C05474=1196.791,200.391,-58.412,-177.682,6.514,148.507
C05475=1196.796,200.142,-58.389,-177.685,6.512,148.508
C05476=1196.800,199.893,-58.365,-177.688,6.510,148.508
C05477=1196.805,199.644,-58.342,-177.690,6.508,148.508
C05478=1196.809,199.396,-58.317,-177.692,6.506,148.509
C05479=1196.813,199.146,-58.294,-177.695,6.505,148.509
C05480=1196.818,198.898,-58.270,-177.698,6.502,148.509
C05481=1196.823,198.649,-58.246,-177.701,6.500,148.510
C05482=1196.827,198.400,-58.222,-177.704,6.498,148.510
C05483=1196.832,198.151,-58.199,-177.706,6.497,148.510
C05484=1196.836,197.902,-58.175,-177.709,6.495,148.511
C05485=1196.841,197.653,-58.151,-177.712,6.493,148.511
C05486=1196.846,197.404,-58.127,-177.714,6.491,148.511
C05487=1196.851,197.155,-58.104,-177.716,6.489,148.511
C05488=1196.855,196.907,-58.080,-177.719,6.487,148.512
C05489=1196.860,196.658,-58.057,-177.722,6.485,148.512
C05490=1196.864,196.409,-58.033,-177.724,6.484,148.512
C05491=1196.869,196.160,-58.009,-177.727,6.482,148.513
C05492=1196.874,195.911,-57.986,-177.730,6.480,148.513
C05493=1196.878,195.662,-57.963,-177.732,6.478,148.514
C05494=1196.883,195.414,-57.938,-177.735,6.476,148.514
C05495=1196.888,195.165,-57.915,-177.738,6.475,148.514
C05496=1196.892,194.916,-57.892,-177.740,6.473,148.515
C05497=1196.896,194.668,-57.868,-177.743,6.471,148.515
C05498=1196.901,194.419,-57.845,-177.745,6.469,148.515
C05499=1196.905,194.170,-57.822,-177.748,6.467,148.515
C05500=1196.910,193.921,-57.798,-177.751,6.465,148.516
C05501=1196.914,193.672,-57.774,-177.753,6.463,148.516
C05502=1196.919,193.423,-57.751,-177.756,6.462,148.516
C05503=1196.924,193.174,-57.727,-177.759,6.460,148.517
C05504=1196.929,192.925,-57.704,-177.761,6.458,148.517
C05505=1196.933,192.676,-57.681,-177.764,6.456,148.517
C05506=1196.938,192.427,-57.657,-177.766,6.454,148.518
C05507=1196.942,192.179,-57.633,-177.769,6.452,148.518
C05508=1196.947,191.930,-57.610,-177.772,6.451,148.519
C05509=1196.951,191.681,-57.587,-177.774,6.449,148.519
C05510=1196.956,191.433,-57.564,-177.777,6.447,148.519
C05511=1196.961,191.184,-57.541,-177.780,6.445,148.520
C05512=1196.966,190.935,-57.517,-177.782,6.443,148.520
C05513=1196.970,190.685,-57.494,-177.785,6.441,148.520
C05514=1196.975,190.436,-57.471,-177.787,6.439,148.520
C05515=1196.979,190.188,-57.448,-177.790,6.438,148.521
C05516=1196.984,189.939,-57.425,-177.793,6.436,148.521
C05517=1196.988,189.690,-57.401,-177.795,6.434,148.521
C05518=1196.993,189.441,-57.378,-177.798,6.432,148.522
C05519=1196.998,189.192,-57.354,-177.801,6.430,148.522
C05520=1197.003,188.943,-57.331,-177.803,6.429,148.523
C05521=1197.007,188.695,-57.309,-177.806,6.427,148.523
C05522=1197.012,188.446,-57.285,-177.809,6.425,148.523
C05523=1197.016,188.196,-57.262,-177.811,6.423,148.524
C05524=1197.021,187.947,-57.239,-177.814,6.421,148.524
C05525=1197.025,187.699,-57.216,-177.817,6.420,148.524
C05526=1197.030,187.450,-57.193,-177.819,6.418,148.525
C05527=1197.035,187.201,-57.169,-177.822,6.416,148.525
C05528=1197.040,186.952,-57.146,-177.825,6.414,148.525
C05529=1197.044,186.704,-57.123,-177.827,6.412,148.526
C05530=1197.049,186.455,-57.100,-177.830,6.411,148.526
C05531=1197.053,186.206,-57.077,-177.833,6.409,148.526
C05532=1197.057,185.957,-57.054,-177.835,6.407,148.527
C05533=1197.062,185.708,-57.031,-177.838,6.405,148.527
C05534=1197.067,185.459,-57.008,-177.841,6.403,148.527
C05535=1197.072,185.189,-56.984,-177.843,6.402,148.528
C05536=1197.077,184.920,-56.958,-177.846,6.400,148.528
C05537=1197.082,184.650,-56.933,-177.849,6.397,148.528
C05538=1197.087,184.381,-56.909,-177.852,6.395,148.529
C05539=1197.092,184.132,-56.885,-177.854,6.394,148.529
C05540=1197.096,183.883,-56.863,-177.857,6.392,148.530
C05541=1197.101,183.634,-56.840,-177.860,6.390,148.530
C05542=1197.105,183.385,-56.817,-177.862,6.388,148.530
C05543=1197.110,183.137,-56.794,-177.864,6.387,148.531
C05544=1197.115,182.887,-56.771,-177.867,6.385,148.531
C05545=1197.120,182.638,-56.748,-177.870,6.384,148.531
C05546=1197.124,182.389,-56.725,-177.872,6.382,148.532
C05547=1197.129,182.140,-56.703,-177.875,6.380,148.532
C05548=1197.133,181.892,-56.680,-177.878,6.378,148.532
C05549=1197.138,181.642,-56.657,-177.880,6.376,148.533
C05550=1197.142,181.394,-56.634,-177.883,6.375,148.533
C05551=1197.147,181.145,-56.612,-177.886,6.373,148.534
C05552=1197.151,180.896,-56.589,-177.888,6.371,148.534
C05553=1197.156,180.647,-56.566,-177.891,6.369,148.534
C05554=1197.161,180.397,-56.543,-177.894,6.367,148.535
C05555=1197.166,180.149,-56.521,-177.896,6.366,148.535
C05556=1197.171,179.900,-56.498,-177.899,6.364,148.535
C05557=1197.175,179.651,-56.475,-177.902,6.362,148.536
C05558=1197.180,179.403,-56.452,-177.904,6.361,148.536
C05559=1197.184,179.153,-56.430,-177.907,6.359,148.537
C05560=1197.189,178.904,-56.407,-177.910,6.358,148.537
C05561=1197.193,178.655,-56.385,-177.912,6.356,148.537
C05562=1197.198,178.407,-56.362,-177.915,6.354,148.538
C05563=1197.203,178.157,-56.340,-177.918,6.352,148.538
C05564=1197.207,177.909,-56.317,-177.920,6.350,148.538
C05565=1197.212,177.660,-56.295,-177.923,6.349,148.539
C05566=1197.216,177.411,-56.272,-177.926,6.347,148.539
C05567=1197.221,177.161,-56.249,-177.928,6.345,148.539
C05568=1197.226,176.913,-56.227,-177.931,6.343,148.540
C05569=1197.231,176.664,-56.204,-177.933,6.342,148.540
C05570=1197.235,176.415,-56.182,-177.936,6.341,148.541
C05571=1197.240,176.166,-56.160,-177.938,6.339,148.541
C05572=1197.244,175.917,-56.137,-177.941,6.337,148.541
C05573=1197.249,175.669,-56.115,-177.944,6.335,148.542
C05574=1197.254,175.419,-56.092,-177.946,6.333,148.542
C05575=1197.258,175.170,-56.069,-177.949,6.332,148.542
C05576=1197.263,174.922,-56.048,-177.952,6.330,148.543
C05577=1197.268,174.672,-56.024,-177.954,6.328,148.543
C05578=1197.272,174.423,-56.002,-177.957,6.326,148.543
C05579=1197.277,174.175,-55.981,-177.959,6.325,148.544
C05580=1197.282,173.925,-55.957,-177.962,6.324,148.544
C05581=1197.286,173.677,-55.936,-177.965,6.322,148.545
C05582=1197.291,173.427,-55.914,-177.968,6.320,148.545
C05583=1197.295,173.178,-55.890,-177.970,6.318,148.546
C05584=1197.300,172.930,-55.869,-177.973,6.317,148.546
C05585=1197.305,172.680,-55.847,-177.976,6.315,148.546
C05586=1197.310,172.432,-55.824,-177.978,6.313,148.547
C05587=1197.314,172.183,-55.801,-177.980,6.312,148.547
C05588=1197.319,171.934,-55.780,-177.983,6.310,148.547
C05589=1197.324,171.685,-55.757,-177.986,6.308,148.548
C05590=1197.328,171.436,-55.734,-177.989,6.307,148.548
C05591=1197.333,171.187,-55.713,-177.991,6.305,148.548
C05592=1197.337,170.938,-55.691,-177.994,6.303,148.549
C05593=1197.343,170.689,-55.668,-177.997,6.301,148.549
C05594=1197.347,170.440,-55.646,-177.999,6.301,148.550
C05595=1197.352,170.192,-55.624,-178.002,6.299,148.550
C05596=1197.356,169.942,-55.602,-178.004,6.297,148.551
C05597=1197.361,169.693,-55.580,-178.007,6.295,148.551
C05598=1197.366,169.444,-55.558,-178.010,6.293,148.551
C05599=1197.371,169.195,-55.536,-178.012,6.292,148.552
C05600=1197.375,168.946,-55.514,-178.015,6.290,148.552
C05601=1197.379,168.698,-55.491,-178.017,6.289,148.552
C05602=1197.384,168.448,-55.469,-178.020,6.287,148.553
C05603=1197.389,168.200,-55.447,-178.023,6.285,148.553
C05604=1197.394,167.950,-55.425,-178.025,6.283,148.553
C05605=1197.398,167.702,-55.403,-178.028,6.282,148.554
C05606=1197.403,167.452,-55.381,-178.031,6.280,148.554
C05607=1197.408,167.204,-55.360,-178.034,6.278,148.555
C05608=1197.413,166.954,-55.337,-178.036,6.277,148.555
C05609=1197.417,166.705,-55.315,-178.039,6.276,148.556
C05610=1197.422,166.456,-55.293,-178.041,6.274,148.556
C05611=1197.427,166.207,-55.272,-178.044,6.272,148.556
C05612=1197.431,165.958,-55.250,-178.047,6.270,148.557
C05613=1197.436,165.709,-55.228,-178.049,6.268,148.557
C05614=1197.440,165.460,-55.206,-178.052,6.268,148.558
C05615=1197.445,165.211,-55.184,-178.054,6.266,148.558
C05616=1197.449,164.962,-55.162,-178.057,6.264,148.558
C05617=1197.455,164.713,-55.140,-178.060,6.262,148.559
C05618=1197.460,164.464,-55.118,-178.062,6.261,148.559
C05619=1197.464,164.215,-55.096,-178.065,6.260,148.559
C05620=1197.469,163.966,-55.074,-178.067,6.258,148.560
C05621=1197.473,163.717,-55.052,-178.070,6.256,148.560
C05622=1197.478,163.468,-55.031,-178.073,6.255,148.561
C05623=1197.482,163.219,-55.009,-178.076,6.253,148.561
C05624=1197.487,162.970,-54.988,-178.078,6.251,148.562
C05625=1197.492,162.721,-54.966,-178.081,6.250,148.562
C05626=1197.496,162.472,-54.944,-178.083,6.248,148.562
C05627=1197.501,162.223,-54.922,-178.086,6.247,148.563
C05628=1197.506,161.974,-54.900,-178.089,6.245,148.563
C05629=1197.510,161.725,-54.878,-178.092,6.243,148.564
C05630=1197.515,161.477,-54.857,-178.094,6.242,148.564
C05631=1197.520,161.227,-54.835,-178.096,6.241,148.564
C05632=1197.525,160.978,-54.814,-178.099,6.239,148.565
C05633=1197.530,160.729,-54.792,-178.102,6.237,148.565
C05634=1197.534,160.480,-54.770,-178.105,6.235,148.566
C05635=1197.539,160.231,-54.749,-178.107,6.234,148.566
C05636=1197.544,159.982,-54.727,-178.110,6.233,148.567
C05637=1197.548,159.733,-54.705,-178.112,6.231,148.567
C05638=1197.552,159.484,-54.684,-178.115,6.229,148.567
C05639=1197.558,159.215,-54.661,-178.118,6.227,148.568
C05640=1197.563,158.946,-54.638,-178.121,6.226,148.568
C05641=1197.568,158.677,-54.614,-178.124,6.224,148.569
C05642=1197.573,158.408,-54.591,-178.126,6.222,148.569
C05643=1197.577,158.160,-54.570,-178.129,6.221,148.569
C05644=1197.582,157.910,-54.548,-178.132,6.220,148.570
C05645=1197.587,157.661,-54.527,-178.134,6.218,148.570
C05646=1197.592,157.412,-54.506,-178.137,6.216,148.571
C05647=1197.596,157.162,-54.484,-178.140,6.215,148.571
C05648=1197.601,156.914,-54.462,-178.142,6.214,148.571
C05649=1197.606,156.665,-54.441,-178.144,6.212,148.572
C05650=1197.610,156.416,-54.420,-178.148,6.210,148.572
C05651=1197.615,156.167,-54.398,-178.150,6.209,148.573
C05652=1197.620,155.918,-54.377,-178.152,6.208,148.573
C05653=1197.625,155.669,-54.355,-178.155,6.206,148.574
C05654=1197.629,155.419,-54.334,-178.158,6.204,148.574
C05655=1197.634,155.170,-54.312,-178.160,6.202,148.574
C05656=1197.639,154.921,-54.292,-178.163,6.202,148.575
C05657=1197.643,154.673,-54.270,-178.166,6.200,148.575
C05658=1197.648,154.423,-54.249,-178.168,6.198,148.576
C05659=1197.653,154.174,-54.227,-178.171,6.196,148.576
C05660=1197.657,153.925,-54.207,-178.173,6.195,148.576
C05661=1197.662,153.677,-54.185,-178.176,6.194,148.577
C05662=1197.667,153.427,-54.164,-178.179,6.192,148.577
C05663=1197.672,153.178,-54.142,-178.182,6.190,148.578
C05664=1197.677,152.929,-54.121,-178.184,6.189,148.578
C05665=1197.681,152.680,-54.100,-178.186,6.188,148.579
C05666=1197.686,152.431,-54.079,-178.190,6.186,148.579
C05667=1197.690,152.182,-54.057,-178.192,6.184,148.580
C05668=1197.695,151.933,-54.037,-178.194,6.184,148.580
C05669=1197.700,151.684,-54.016,-178.197,6.182,148.580
C05670=1197.705,151.435,-53.994,-178.200,6.180,148.581
C05671=1197.710,151.186,-53.973,-178.203,6.178,148.581
C05672=1197.714,150.937,-53.951,-178.205,6.178,148.582
C05673=1197.719,150.687,-53.931,-178.208,6.176,148.582
C05674=1197.724,150.438,-53.910,-178.210,6.174,148.582
C05675=1197.728,150.190,-53.888,-178.213,6.172,148.583
C05676=1197.733,149.941,-53.868,-178.216,6.172,148.583
C05677=1197.738,149.691,-53.847,-178.218,6.170,148.584
C05678=1197.742,149.442,-53.825,-178.221,6.168,148.584
C05679=1197.747,149.193,-53.804,-178.223,6.167,148.585
C05680=1197.752,148.944,-53.784,-178.226,6.166,148.585
C05681=1197.757,148.695,-53.763,-178.229,6.164,148.586
C05682=1197.762,148.446,-53.741,-178.232,6.162,148.586
C05683=1197.766,148.197,-53.721,-178.234,6.161,148.586
C05684=1197.771,147.948,-53.700,-178.237,6.160,148.587
C05685=1197.775,147.698,-53.679,-178.240,6.158,148.587
C05686=1197.780,147.450,-53.657,-178.242,6.157,148.588
C05687=1197.785,147.200,-53.636,-178.244,6.155,148.588
C05688=1197.790,146.951,-53.616,-178.247,6.153,148.588
C05689=1197.795,146.702,-53.595,-178.250,6.152,148.589
C05690=1197.799,146.454,-53.574,-178.252,6.151,148.589
C05691=1197.804,146.205,-53.553,-178.255,6.149,148.590
C05692=1197.808,145.956,-53.533,-178.258,6.147,148.590
C05693=1197.814,145.706,-53.512,-178.260,6.147,148.591
C05694=1197.818,145.456,-53.490,-178.263,6.145,148.591
C05695=1197.823,145.207,-53.470,-178.266,6.143,148.592
C05696=1197.828,144.958,-53.449,-178.268,6.142,148.592
C05697=1197.832,144.710,-53.428,-178.271,6.141,148.593
C05698=1197.837,144.461,-53.407,-178.274,6.139,148.593
C05699=1197.842,144.212,-53.387,-178.276,6.138,148.593
C05700=1197.847,143.962,-53.366,-178.278,6.136,148.594
C05701=1197.851,143.713,-53.345,-178.282,6.135,148.594
C05702=1197.856,143.465,-53.325,-178.284,6.133,148.595
C05703=1197.861,143.215,-53.304,-178.286,6.132,148.595
C05704=1197.865,142.966,-53.283,-178.289,6.130,148.596
C05705=1197.870,142.717,-53.263,-178.292,6.129,148.596
C05706=1197.875,142.468,-53.242,-178.294,6.128,148.597
C05707=1197.880,142.219,-53.221,-178.297,6.126,148.597
C05708=1197.884,141.970,-53.201,-178.300,6.124,148.597
C05709=1197.890,141.721,-53.180,-178.302,6.124,148.598
C05710=1197.894,141.472,-53.159,-178.305,6.122,148.598
C05711=1197.898,141.222,-53.139,-178.308,6.120,148.599
C05712=1197.903,140.973,-53.118,-178.310,6.120,148.599
C05713=1197.908,140.724,-53.097,-178.313,6.118,148.600
C05714=1197.913,140.475,-53.076,-178.316,6.116,148.600
C05715=1197.917,140.226,-53.056,-178.318,6.115,148.601
C05716=1197.922,139.977,-53.036,-178.321,6.114,148.601
C05717=1197.927,139.727,-53.015,-178.324,6.112,148.602
C05718=1197.931,139.478,-52.994,-178.326,6.111,148.602
C05719=1197.936,139.230,-52.974,-178.329,6.110,148.603
C05720=1197.942,138.980,-52.954,-178.332,6.108,148.603
C05721=1197.946,138.731,-52.934,-178.334,6.107,148.603
C05722=1197.951,138.482,-52.913,-178.336,6.105,148.604
C05723=1197.956,138.233,-52.892,-178.339,6.105,148.604
C05724=1197.960,137.984,-52.872,-178.342,6.103,148.605
C05725=1197.965,137.735,-52.852,-178.344,6.101,148.605
C05726=1197.970,137.486,-52.831,-178.347,6.100,148.606
C05727=1197.975,137.236,-52.811,-178.350,6.099,148.606
C05728=1197.979,136.988,-52.791,-178.352,6.097,148.606
C05729=1197.984,136.738,-52.770,-178.354,6.096,148.607
C05730=1197.989,136.489,-52.749,-178.358,6.094,148.608
C05731=1197.993,136.240,-52.730,-178.360,6.093,148.608
C05732=1197.998,135.991,-52.709,-178.362,6.092,148.608
C05733=1198.003,135.742,-52.688,-178.366,6.090,148.609
C05734=1198.007,135.493,-52.668,-178.368,6.089,148.609
C05735=1198.012,135.243,-52.648,-178.370,6.088,148.610
C05736=1198.017,134.994,-52.628,-178.374,6.086,148.610
C05737=1198.022,134.745,-52.607,-178.376,6.085,148.611
C05738=1198.027,134.497,-52.587,-178.378,6.083,148.611
C05739=1198.032,134.247,-52.567,-178.382,6.082,148.612
C05740=1198.036,133.998,-52.547,-178.384,6.081,148.612
C05741=1198.040,133.749,-52.527,-178.386,6.079,148.613
C05742=1198.046,133.499,-52.506,-178.388,6.078,148.613
C05743=1198.050,133.231,-52.484,-178.392,6.077,148.614
C05744=1198.056,132.962,-52.463,-178.394,6.075,148.614
C05745=1198.061,132.694,-52.441,-178.398,6.074,148.615
C05746=1198.066,132.425,-52.419,-178.400,6.072,148.615
C05747=1198.071,132.176,-52.399,-178.403,6.071,148.616
C05748=1198.076,131.927,-52.379,-178.406,6.070,148.616
C05749=1198.080,131.678,-52.359,-178.408,6.068,148.616
C05750=1198.085,131.428,-52.339,-178.411,6.067,148.617
C05751=1198.091,131.180,-52.319,-178.413,6.065,148.617
C05752=1198.095,130.930,-52.299,-178.416,6.064,148.618
C05753=1198.100,130.681,-52.279,-178.419,6.063,148.618
C05754=1198.104,130.432,-52.259,-178.421,6.061,148.619
C05755=1198.109,130.183,-52.239,-178.424,6.060,148.619
C05756=1198.113,129.934,-52.218,-178.427,6.059,148.620
C05757=1198.119,129.685,-52.199,-178.429,6.058,148.620
C05758=1198.123,129.436,-52.179,-178.432,6.056,148.621
C05759=1198.128,129.186,-52.159,-178.435,6.055,148.621
C05760=1198.133,128.936,-52.139,-178.437,6.054,148.622
C05761=1198.138,128.687,-52.118,-178.440,6.052,148.622
C05762=1198.143,128.439,-52.099,-178.442,6.051,148.623
C05763=1198.148,128.190,-52.079,-178.445,6.050,148.623
C05764=1198.152,127.940,-52.059,-178.447,6.049,148.624
C05765=1198.157,127.691,-52.039,-178.450,6.047,148.624
C05766=1198.162,127.442,-52.019,-178.453,6.046,148.624
C05767=1198.167,127.193,-51.999,-178.455,6.045,148.625
C05768=1198.171,126.944,-51.979,-178.458,6.043,148.625
C05769=1198.176,126.694,-51.960,-178.460,6.042,148.626
C05770=1198.180,126.445,-51.939,-178.463,6.041,148.626
C05771=1198.186,126.196,-51.920,-178.466,6.040,148.627
C05772=1198.191,125.947,-51.900,-178.468,6.038,148.627
C05773=1198.195,125.698,-51.880,-178.471,6.037,148.628
C05774=1198.200,125.448,-51.860,-178.474,6.036,148.628
C05775=1198.205,125.199,-51.841,-178.477,6.034,148.629
C05776=1198.209,124.950,-51.821,-178.479,6.033,148.629
C05777=1198.214,124.701,-51.801,-178.482,6.032,148.630
C05778=1198.220,124.452,-51.782,-178.484,6.031,148.630
C05779=1198.224,124.203,-51.761,-178.487,6.029,148.631
C05780=1198.228,123.954,-51.742,-178.490,6.028,148.631
C05781=1198.233,123.704,-51.723,-178.492,6.027,148.632
C05782=1198.238,123.455,-51.703,-178.495,6.025,148.632
C05783=1198.243,123.206,-51.683,-178.497,6.024,148.633
C05784=1198.247,122.957,-51.663,-178.500,6.023,148.633
C05785=1198.253,122.708,-51.644,-178.502,6.022,148.634
C05786=1198.257,122.458,-51.624,-178.505,6.020,148.634
C05787=1198.262,122.209,-51.604,-178.508,6.020,148.635
C05788=1198.267,121.961,-51.585,-178.510,6.018,148.635
C05789=1198.272,121.711,-51.565,-178.513,6.017,148.636
C05790=1198.276,121.462,-51.546,-178.516,6.015,148.636
C05791=1198.281,121.213,-51.527,-178.519,6.014,148.637
C05792=1198.286,120.963,-51.507,-178.521,6.013,148.637
C05793=1198.290,120.714,-51.487,-178.524,6.011,148.637
C05794=1198.296,120.466,-51.467,-178.526,6.011,148.638
C05795=1198.300,120.216,-51.448,-178.529,6.009,148.639
C05796=1198.305,119.967,-51.429,-178.531,6.008,148.639
C05797=1198.310,119.718,-51.409,-178.534,6.007,148.640
C05798=1198.315,119.468,-51.390,-178.536,6.006,148.640
C05799=1198.319,119.219,-51.370,-178.539,6.004,148.641
C05800=1198.325,118.970,-51.351,-178.542,6.003,148.641
C05801=1198.329,118.720,-51.331,-178.545,6.002,148.642
C05802=1198.334,118.472,-51.312,-178.547,6.001,148.642
C05803=1198.338,118.223,-51.292,-178.550,5.999,148.642
C05804=1198.343,117.973,-51.272,-178.552,5.999,148.643
C05805=1198.349,117.724,-51.253,-178.555,5.997,148.643
C05806=1198.353,117.475,-51.234,-178.557,5.996,148.644
C05807=1198.357,117.225,-51.214,-178.560,5.994,148.645
C05808=1198.363,116.977,-51.195,-178.562,5.994,148.645
C05809=1198.367,116.727,-51.175,-178.566,5.992,148.646
C05810=1198.372,116.478,-51.157,-178.568,5.990,148.646
C05811=1198.377,116.229,-51.137,-178.571,5.990,148.647
C05812=1198.382,115.980,-51.118,-178.574,5.988,148.647
C05813=1198.387,115.730,-51.099,-178.576,5.987,148.647
C05814=1198.391,115.481,-51.080,-178.579,5.986,148.648
C05815=1198.396,115.232,-51.060,-178.581,5.985,148.648
C05816=1198.401,114.982,-51.041,-178.584,5.983,148.649
C05817=1198.406,114.734,-51.022,-178.586,5.982,148.649
C05818=1198.411,114.484,-51.002,-178.589,5.981,148.650
C05819=1198.416,114.235,-50.983,-178.592,5.980,148.651
C05820=1198.420,113.986,-50.964,-178.594,5.978,148.651
C05821=1198.425,113.737,-50.945,-178.597,5.978,148.652
C05822=1198.430,113.487,-50.925,-178.600,5.976,148.652
C05823=1198.435,113.238,-50.907,-178.602,5.975,148.653
C05824=1198.440,112.989,-50.888,-178.604,5.974,148.653
C05825=1198.445,112.740,-50.868,-178.607,5.973,148.654
C05826=1198.449,112.491,-50.849,-178.610,5.972,148.654
C05827=1198.454,112.242,-50.830,-178.612,5.970,148.654
C05828=1198.459,111.992,-50.810,-178.615,5.970,148.655
C05829=1198.464,111.743,-50.792,-178.618,5.968,148.655
C05830=1198.469,111.493,-50.773,-178.620,5.967,148.656
C05831=1198.473,111.245,-50.754,-178.623,5.966,148.657
C05832=1198.478,110.995,-50.734,-178.626,5.965,148.657
C05833=1198.483,110.746,-50.716,-178.628,5.963,148.658
C05834=1198.488,110.497,-50.697,-178.631,5.963,148.658
C05835=1198.493,110.248,-50.677,-178.634,5.961,148.659
C05836=1198.497,109.998,-50.658,-178.636,5.960,148.659
C05837=1198.503,109.749,-50.640,-178.639,5.959,148.660
C05838=1198.507,109.500,-50.621,-178.641,5.958,148.660
C05839=1198.512,109.251,-50.601,-178.644,5.956,148.661
C05840=1198.516,109.001,-50.583,-178.646,5.955,148.661
C05841=1198.522,108.752,-50.564,-178.649,5.954,148.662
C05842=1198.526,108.503,-50.545,-178.652,5.953,148.662
C05843=1198.531,108.253,-50.526,-178.654,5.952,148.663
C05844=1198.536,108.005,-50.507,-178.657,5.951,148.663
C05845=1198.541,107.755,-50.488,-178.660,5.950,148.664
C05846=1198.546,107.506,-50.470,-178.662,5.948,148.664
C05847=1198.551,107.237,-50.449,-178.665,5.948,148.665
C05848=1198.556,106.969,-50.429,-178.668,5.946,148.665
C05849=1198.561,106.701,-50.408,-178.671,5.945,148.666
C05850=1198.566,106.432,-50.388,-178.673,5.944,148.667
C05851=1198.572,106.183,-50.369,-178.676,5.942,148.667
C05852=1198.576,105.934,-50.350,-178.679,5.942,148.668
C05853=1198.581,105.685,-50.332,-178.681,5.940,148.668
C05854=1198.586,105.436,-50.312,-178.684,5.939,148.669
C05855=1198.590,105.186,-50.294,-178.687,5.938,148.669
C05856=1198.596,104.937,-50.275,-178.689,5.937,148.670
C05857=1198.600,104.687,-50.257,-178.691,5.936,148.670
C05858=1198.605,104.438,-50.237,-178.694,5.934,148.671
C05859=1198.610,104.189,-50.219,-178.697,5.934,148.671
C05860=1198.614,103.940,-50.200,-178.699,5.932,148.672
C05861=1198.620,103.690,-50.182,-178.702,5.931,148.672
C05862=1198.624,103.442,-50.163,-178.705,5.930,148.673
C05863=1198.629,103.192,-50.145,-178.707,5.929,148.673
C05864=1198.634,102.943,-50.125,-178.710,5.928,148.674
C05865=1198.638,102.693,-50.107,-178.713,5.927,148.674
C05866=1198.644,102.444,-50.088,-178.715,5.926,148.675
C05867=1198.649,102.195,-50.070,-178.718,5.925,148.675
C05868=1198.653,101.945,-50.051,-178.720,5.924,148.676
C05869=1198.658,101.696,-50.032,-178.723,5.922,148.676
C05870=1198.663,101.447,-50.014,-178.725,5.921,148.677
C05871=1198.667,101.198,-49.995,-178.728,5.921,148.678
C05872=1198.673,100.948,-49.976,-178.731,5.919,148.678
C05873=1198.678,100.699,-49.958,-178.733,5.918,148.679
C05874=1198.682,100.451,-49.940,-178.736,5.917,148.679
C05875=1198.687,100.201,-49.921,-178.739,5.916,148.680
C05876=1198.692,99.951,-49.903,-178.741,5.915,148.680
C05877=1198.697,99.703,-49.884,-178.744,5.914,148.681
C05878=1198.701,99.453,-49.866,-178.746,5.913,148.681
C05879=1198.707,99.203,-49.847,-178.749,5.911,148.682
C05880=1198.712,98.955,-49.829,-178.752,5.910,148.682
C05881=1198.716,98.705,-49.810,-178.754,5.910,148.683
C05882=1198.721,98.456,-49.792,-178.757,5.908,148.683
C05883=1198.726,98.206,-49.774,-178.759,5.908,148.684
C05884=1198.731,97.958,-49.755,-178.762,5.906,148.684
C05885=1198.735,97.708,-49.737,-178.765,5.905,148.685
C05886=1198.740,97.459,-49.719,-178.767,5.904,148.685
C05887=1198.746,97.209,-49.700,-178.770,5.903,148.686
C05888=1198.751,96.961,-49.681,-178.772,5.902,148.686
C05889=1198.755,96.711,-49.663,-178.775,5.901,148.687
C05890=1198.760,96.462,-49.645,-178.778,5.900,148.687
C05891=1198.765,96.212,-49.627,-178.780,5.899,148.688
C05892=1198.770,95.963,-49.608,-178.783,5.898,148.689
C05893=1198.774,95.714,-49.589,-178.786,5.897,148.689
C05894=1198.779,95.465,-49.571,-178.789,5.895,148.690
C05895=1198.784,95.215,-49.553,-178.791,5.894,148.690
C05896=1198.789,94.966,-49.535,-178.793,5.894,148.691
C05897=1198.794,94.717,-49.517,-178.796,5.892,148.691
C05898=1198.799,94.467,-49.499,-178.799,5.892,148.692
C05899=1198.804,94.218,-49.481,-178.801,5.891,148.692
C05900=1198.809,93.969,-49.462,-178.804,5.889,148.693
C05901=1198.813,93.720,-49.444,-178.806,5.888,148.693
C05902=1198.818,93.471,-49.426,-178.809,5.887,148.694
C05903=1198.823,93.221,-49.408,-178.812,5.886,148.694
C05904=1198.828,92.972,-49.390,-178.814,5.885,148.695
C05905=1198.833,92.723,-49.372,-178.817,5.884,148.696
C05906=1198.838,92.473,-49.353,-178.820,5.883,148.696
C05907=1198.843,92.224,-49.335,-178.822,5.883,148.697
C05908=1198.848,91.975,-49.317,-178.825,5.881,148.697
C05909=1198.852,91.725,-49.299,-178.827,5.880,148.698
C05910=1198.857,91.476,-49.281,-178.830,5.879,148.698
C05911=1198.862,91.226,-49.263,-178.833,5.878,148.699
C05912=1198.867,90.977,-49.245,-178.835,5.877,148.699
C05913=1198.872,90.728,-49.227,-178.838,5.876,148.700
C05914=1198.877,90.479,-49.209,-178.840,5.875,148.700
C05915=1198.881,90.229,-49.190,-178.843,5.874,148.701
C05916=1198.886,89.980,-49.172,-178.846,5.872,148.702
C05917=1198.891,89.731,-49.154,-178.848,5.872,148.702
C05918=1198.896,89.482,-49.137,-178.851,5.871,148.703
C05919=1198.901,89.232,-49.119,-178.854,5.870,148.703
C05920=1198.906,88.983,-49.101,-178.856,5.869,148.704
C05921=1198.911,88.734,-49.083,-178.858,5.868,148.704
C05922=1198.916,88.485,-49.065,-178.862,5.867,148.705
C05923=1198.920,88.236,-49.047,-178.864,5.866,148.705
C05924=1198.925,87.985,-49.029,-178.866,5.865,148.706
C05925=1198.930,87.736,-49.011,-178.869,5.863,148.706
C05926=1198.935,87.487,-48.993,-178.872,5.863,148.707
C05927=1198.940,87.238,-48.975,-178.874,5.862,148.708
C05928=1198.945,86.988,-48.957,-178.877,5.861,148.708
C05929=1198.950,86.739,-48.939,-178.880,5.860,148.709
C05930=1198.955,86.490,-48.921,-178.882,5.859,148.709
C05931=1198.960,86.240,-48.904,-178.885,5.858,148.710
C05932=1198.965,85.991,-48.886,-178.887,5.857,148.710
C05933=1198.970,85.742,-48.868,-178.890,5.856,148.711
C05934=1198.975,85.493,-48.850,-178.893,5.855,148.712
C05935=1198.979,85.244,-48.833,-178.895,5.854,148.712
C05936=1198.984,84.994,-48.815,-178.898,5.853,148.713
C05937=1198.988,84.744,-48.797,-178.900,5.852,148.713
C05938=1198.993,84.495,-48.779,-178.903,5.851,148.714
C05939=1198.998,84.246,-48.761,-178.905,5.850,148.714
C05940=1199.003,83.996,-48.744,-178.908,5.850,148.715
C05941=1199.008,83.747,-48.726,-178.911,5.848,148.715
C05942=1199.013,83.498,-48.708,-178.913,5.847,148.716
C05943=1199.018,83.249,-48.690,-178.916,5.847,148.717
C05944=1199.022,82.999,-48.673,-178.918,5.845,148.717
C05945=1199.027,82.750,-48.655,-178.921,5.844,148.718
C05946=1199.032,82.501,-48.637,-178.924,5.844,148.718
C05947=1199.038,82.251,-48.620,-178.926,5.842,148.719
C05948=1199.042,82.002,-48.602,-178.929,5.842,148.719
C05949=1199.047,81.753,-48.584,-178.931,5.841,148.720
C05950=1199.052,81.503,-48.567,-178.934,5.840,148.720
C05951=1199.057,81.235,-48.548,-178.937,5.839,148.721
C05952=1199.063,80.967,-48.529,-178.939,5.838,148.722
C05953=1199.068,80.698,-48.510,-178.942,5.836,148.722
C05954=1199.073,80.430,-48.491,-178.945,5.836,148.723
C05955=1199.078,80.180,-48.473,-178.948,5.835,148.723
C05956=1199.082,79.932,-48.456,-178.950,5.834,148.724
C05957=1199.088,79.682,-48.439,-178.953,5.833,148.725
C05958=1199.093,79.433,-48.421,-178.955,5.832,148.725
C05959=1199.098,79.183,-48.403,-178.958,5.831,148.726
C05960=1199.102,78.934,-48.386,-178.961,5.830,148.726
C05961=1199.107,78.684,-48.369,-178.963,5.829,148.727
C05962=1199.112,78.435,-48.351,-178.966,5.828,148.727
C05963=1199.117,78.185,-48.334,-178.968,5.827,148.728
C05964=1199.122,77.937,-48.317,-178.971,5.826,148.728
C05965=1199.127,77.687,-48.299,-178.974,5.826,148.729
C05966=1199.132,77.438,-48.281,-178.976,5.824,148.730
C05967=1199.137,77.188,-48.264,-178.979,5.824,148.730
C05968=1199.142,76.939,-48.247,-178.981,5.823,148.731
C05969=1199.147,76.690,-48.229,-178.984,5.821,148.731
C05970=1199.152,76.440,-48.211,-178.987,5.821,148.732
C05971=1199.156,76.191,-48.195,-178.989,5.820,148.732
C05972=1199.161,75.942,-48.177,-178.992,5.819,148.733
C05973=1199.166,75.692,-48.160,-178.995,5.818,148.734
C05974=1199.171,75.443,-48.142,-178.997,5.817,148.734
C05975=1199.176,75.194,-48.125,-179.000,5.816,148.735
C05976=1199.182,74.944,-48.108,-179.002,5.816,148.735
C05977=1199.186,74.695,-48.091,-179.005,5.814,148.736
C05978=1199.191,74.445,-48.073,-179.008,5.814,148.736
C05979=1199.195,74.197,-48.056,-179.010,5.813,148.737
C05980=1199.200,73.947,-48.039,-179.012,5.812,148.738
C05981=1199.206,73.697,-48.021,-179.015,5.810,148.738
C05982=1199.210,73.448,-48.004,-179.018,5.810,148.739
C05983=1199.216,73.199,-47.987,-179.020,5.809,148.739
C05984=1199.220,72.950,-47.970,-179.022,5.808,148.740
C05985=1199.225,72.700,-47.952,-179.026,5.807,148.740
C05986=1199.230,72.451,-47.935,-179.028,5.806,148.741
C05987=1199.235,72.201,-47.919,-179.030,5.806,148.741
C05988=1199.240,71.952,-47.901,-179.033,5.805,148.742
C05989=1199.245,71.703,-47.884,-179.036,5.804,148.743
C05990=1199.250,71.453,-47.867,-179.038,5.803,148.743
C05991=1199.254,71.204,-47.850,-179.041,5.802,148.744
C05992=1199.259,70.955,-47.832,-179.043,5.801,148.744
C05993=1199.264,70.705,-47.815,-179.046,5.800,148.745
C05994=1199.269,70.455,-47.798,-179.049,5.799,148.746
C05995=1199.275,70.206,-47.782,-179.051,5.798,148.746
C05996=1199.279,69.957,-47.764,-179.054,5.798,148.747
C05997=1199.284,69.708,-47.747,-179.056,5.797,148.747
C05998=1199.289,69.458,-47.730,-179.059,5.796,148.748
C05999=1199.294,69.208,-47.713,-179.062,5.795,148.748
C06000=1199.299,68.960,-47.697,-179.064,5.794,148.749
C06001=1199.304,68.710,-47.679,-179.067,5.794,148.750
C06002=1199.308,68.461,-47.662,-179.070,5.792,148.750
C06003=1199.314,68.211,-47.645,-179.072,5.791,148.751
C06004=1199.319,67.962,-47.628,-179.075,5.791,148.751
C06005=1199.323,67.713,-47.612,-179.077,5.790,148.752
C06006=1199.328,67.463,-47.594,-179.079,5.789,148.752
C06007=1199.333,67.214,-47.578,-179.083,5.788,148.753
C06008=1199.338,66.965,-47.560,-179.085,5.787,148.754
C06009=1199.343,66.716,-47.544,-179.087,5.786,148.754
C06010=1199.348,66.466,-47.526,-179.090,5.786,148.755
C06011=1199.352,66.216,-47.510,-179.093,5.785,148.755
C06012=1199.358,65.967,-47.493,-179.095,5.784,148.756
C06013=1199.363,65.718,-47.476,-179.098,5.783,148.757
C06014=1199.367,65.468,-47.459,-179.101,5.783,148.757
C06015=1199.372,65.219,-47.442,-179.103,5.782,148.758
C06016=1199.378,64.970,-47.426,-179.106,5.780,148.758
C06017=1199.383,64.720,-47.409,-179.109,5.780,148.759
C06018=1199.387,64.470,-47.392,-179.111,5.779,148.759
C06019=1199.392,64.221,-47.375,-179.113,5.778,148.760
C06020=1199.398,63.972,-47.358,-179.116,5.778,148.761
C06021=1199.402,63.722,-47.342,-179.119,5.776,148.761
C06022=1199.407,63.473,-47.325,-179.121,5.775,148.762
C06023=1199.412,63.224,-47.308,-179.124,5.775,148.763
C06024=1199.417,62.974,-47.291,-179.126,5.774,148.763
C06025=1199.421,62.725,-47.275,-179.129,5.773,148.764
C06026=1199.427,62.476,-47.258,-179.132,5.772,148.764
C06027=1199.432,62.226,-47.241,-179.134,5.771,148.765
C06028=1199.436,61.977,-47.224,-179.137,5.771,148.765
C06029=1199.442,61.728,-47.208,-179.139,5.770,148.766
C06030=1199.446,61.478,-47.191,-179.141,5.769,148.766
C06031=1199.451,61.229,-47.174,-179.144,5.769,148.767
C06032=1199.457,60.980,-47.157,-179.147,5.767,148.768
C06033=1199.461,60.730,-47.141,-179.149,5.766,148.768
C06034=1199.466,60.480,-47.125,-179.152,5.766,148.769
C06035=1199.471,60.231,-47.108,-179.155,5.765,148.770
C06036=1199.476,59.981,-47.091,-179.157,5.764,148.770
C06037=1199.481,59.732,-47.074,-179.160,5.763,148.771
C06038=1199.486,59.483,-47.058,-179.163,5.763,148.771
C06039=1199.490,59.234,-47.042,-179.165,5.762,148.772
C06040=1199.496,58.984,-47.025,-179.167,5.761,148.772
C06041=1199.501,58.735,-47.009,-179.170,5.761,148.773
C06042=1199.505,58.485,-46.992,-179.172,5.760,148.774
C06043=1199.510,58.236,-46.976,-179.175,5.758,148.774
C06044=1199.516,57.986,-46.958,-179.178,5.758,148.775
C06045=1199.521,57.737,-46.943,-179.180,5.757,148.775
C06046=1199.526,57.488,-46.926,-179.183,5.756,148.776
C06047=1199.530,57.238,-46.910,-179.186,5.756,148.777
C06048=1199.535,56.989,-46.893,-179.188,5.755,148.777
C06049=1199.540,56.740,-46.876,-179.191,5.754,148.778
C06050=1199.546,56.490,-46.860,-179.194,5.753,148.778
C06051=1199.550,56.241,-46.844,-179.196,5.752,148.779
C06052=1199.555,55.991,-46.827,-179.198,5.752,148.779
C06053=1199.560,55.742,-46.811,-179.201,5.751,148.780
C06054=1199.565,55.492,-46.794,-179.204,5.750,148.781
C06055=1199.571,55.224,-46.776,-179.207,5.749,148.781
C06056=1199.576,54.956,-46.759,-179.209,5.748,148.782
C06057=1199.581,54.687,-46.741,-179.212,5.748,148.783
C06058=1199.586,54.419,-46.724,-179.215,5.746,148.783
C06059=1199.591,54.169,-46.708,-179.217,5.746,148.784
C06060=1199.597,53.919,-46.691,-179.220,5.745,148.785
C06061=1199.601,53.670,-46.675,-179.222,5.744,148.785
C06062=1199.606,53.421,-46.658,-179.225,5.744,148.786
C06063=1199.611,53.171,-46.643,-179.227,5.743,148.786
C06064=1199.616,52.922,-46.626,-179.230,5.742,148.787
C06065=1199.621,52.672,-46.610,-179.232,5.742,148.787
C06066=1199.626,52.423,-46.594,-179.235,5.740,148.788
C06067=1199.631,52.174,-46.577,-179.238,5.740,148.789
C06068=1199.636,51.924,-46.562,-179.240,5.739,148.789
C06069=1199.641,51.675,-46.545,-179.243,5.739,148.790
C06070=1199.646,51.426,-46.529,-179.246,5.738,148.791
C06071=1199.650,51.176,-46.513,-179.248,5.737,148.791
C06072=1199.657,50.926,-46.497,-179.250,5.737,148.792
C06073=1199.661,50.677,-46.480,-179.254,5.735,148.792
C06074=1199.666,50.428,-46.464,-179.256,5.735,148.793
C06075=1199.671,50.178,-46.448,-179.258,5.734,148.793
C06076=1199.676,49.929,-46.431,-179.261,5.733,148.794
C06077=1199.681,49.679,-46.415,-179.264,5.733,148.795
C06078=1199.686,49.430,-46.399,-179.266,5.732,148.795
C06079=1199.691,49.180,-46.383,-179.268,5.731,148.796
C06080=1199.696,48.931,-46.367,-179.271,5.731,148.797
C06081=1199.700,48.681,-46.351,-179.274,5.730,148.797
C06082=1199.706,48.432,-46.335,-179.276,5.728,148.798
C06083=1199.710,48.182,-46.319,-179.279,5.728,148.798
C06084=1199.716,47.933,-46.303,-179.282,5.727,148.799
C06085=1199.719,47.684,-46.287,-179.284,5.727,148.799
C06086=1199.725,47.434,-46.271,-179.286,5.726,148.800
C06087=1199.730,47.186,-46.255,-179.289,5.725,148.801
C06088=1199.735,46.936,-46.239,-179.292,5.725,148.801
C06089=1199.740,46.686,-46.224,-179.294,5.724,148.802
C06090=1199.745,46.437,-46.207,-179.297,5.724,148.803
C06091=1199.750,46.187,-46.191,-179.300,5.722,148.803
C06092=1199.754,45.938,-46.175,-179.302,5.722,148.804
C06093=1199.760,45.688,-46.159,-179.305,5.721,148.804
C06094=1199.765,45.439,-46.143,-179.307,5.720,148.805
C06095=1199.770,45.190,-46.127,-179.310,5.720,148.806
C06096=1199.775,44.940,-46.111,-179.312,5.719,148.806
C06097=1199.780,44.690,-46.095,-179.315,5.718,148.807
C06098=1199.784,44.442,-46.080,-179.317,5.718,148.808
C06099=1199.790,44.192,-46.064,-179.320,5.717,148.808
C06100=1199.794,43.942,-46.048,-179.322,5.716,148.809
C06101=1199.800,43.693,-46.032,-179.325,5.716,148.809
C06102=1199.805,43.444,-46.016,-179.328,5.714,148.810
C06103=1199.810,43.194,-46.000,-179.331,5.714,148.811
C06104=1199.815,42.944,-45.985,-179.333,5.713,148.811
C06105=1199.820,42.695,-45.968,-179.335,5.712,148.812
C06106=1199.824,42.446,-45.953,-179.338,5.712,148.812
C06107=1199.830,42.196,-45.937,-179.340,5.711,148.813
C06108=1199.834,41.946,-45.921,-179.343,5.711,148.814
C06109=1199.840,41.697,-45.906,-179.345,5.710,148.814
C06110=1199.845,41.448,-45.889,-179.348,5.709,148.815
C06111=1199.850,41.198,-45.873,-179.350,5.709,148.815
C06112=1199.854,40.949,-45.859,-179.353,5.708,148.816
C06113=1199.860,40.699,-45.843,-179.355,5.708,148.817
C06114=1199.864,40.449,-45.827,-179.358,5.707,148.817
C06115=1199.869,40.201,-45.811,-179.361,5.705,148.818
C06116=1199.874,39.952,-45.796,-179.363,5.705,148.818
C06117=1199.879,39.701,-45.780,-179.366,5.704,148.819
C06118=1199.884,39.452,-45.764,-179.369,5.704,148.820
C06119=1199.890,39.203,-45.749,-179.371,5.703,148.820
C06120=1199.894,38.952,-45.733,-179.374,5.702,148.821
C06121=1199.899,38.703,-45.718,-179.376,5.702,148.822
C06122=1199.904,38.455,-45.701,-179.379,5.701,148.822
C06123=1199.910,38.205,-45.686,-179.381,5.700,148.823
C06124=1199.914,37.955,-45.670,-179.384,5.700,148.823
C06125=1199.919,37.706,-45.655,-179.386,5.699,148.824
C06126=1199.924,37.457,-45.639,-179.389,5.699,148.825
C06127=1199.930,37.207,-45.624,-179.391,5.698,148.825
C06128=1199.934,36.957,-45.608,-179.394,5.697,148.826
C06129=1199.939,36.708,-45.593,-179.396,5.697,148.827
C06130=1199.945,36.459,-45.577,-179.399,5.696,148.827
C06131=1199.949,36.209,-45.561,-179.401,5.695,148.828
C06132=1199.954,35.959,-45.546,-179.404,5.694,148.828
C06133=1199.959,35.710,-45.531,-179.407,5.694,148.829
C06134=1199.965,35.461,-45.515,-179.410,5.693,148.830
C06135=1199.969,35.211,-45.500,-179.412,5.692,148.830
C06136=1199.974,34.961,-45.484,-179.414,5.692,148.831
C06137=1199.980,34.712,-45.468,-179.417,5.691,148.831
C06138=1199.984,34.463,-45.453,-179.420,5.691,148.832
C06139=1199.990,34.214,-45.438,-179.422,5.690,148.833
C06140=1199.994,33.964,-45.422,-179.425,5.689,148.833
C06141=1199.999,33.714,-45.407,-179.427,5.689,148.834
C06142=1200.005,33.465,-45.391,-179.430,5.688,148.835
C06143=1200.009,33.216,-45.376,-179.432,5.688,148.835
C06144=1200.014,32.966,-45.360,-179.435,5.687,148.836
C06145=1200.019,32.716,-45.345,-179.437,5.686,148.836
C06146=1200.024,32.467,-45.330,-179.440,5.686,148.837
C06147=1200.029,32.218,-45.314,-179.443,5.685,148.838
C06148=1200.034,31.968,-45.300,-179.445,5.684,148.838
C06149=1200.039,31.718,-45.284,-179.447,5.684,148.839
C06150=1200.045,31.469,-45.268,-179.450,5.683,148.840
C06151=1200.049,31.220,-45.253,-179.453,5.683,148.840
C06152=1200.055,30.970,-45.238,-179.455,5.682,148.841
C06153=1200.059,30.721,-45.223,-179.457,5.681,148.841
C06154=1200.065,30.472,-45.207,-179.460,5.681,148.842
C06155=1200.069,30.221,-45.193,-179.463,5.680,148.843
C06156=1200.074,29.972,-45.177,-179.465,5.679,148.843
C06157=1200.079,29.723,-45.162,-179.468,5.679,148.844
C06158=1200.084,29.473,-45.146,-179.470,5.678,148.845
C06159=1200.089,29.205,-45.131,-179.473,5.678,148.845
C06160=1200.095,28.936,-45.114,-179.476,5.677,148.846
C06161=1200.101,28.667,-45.097,-179.479,5.676,148.847
C06162=1200.106,28.399,-45.081,-179.481,5.676,148.847
C06163=1200.111,28.149,-45.066,-179.484,5.675,148.848
C06164=1200.115,27.899,-45.051,-179.487,5.675,148.849
C06165=1200.121,27.650,-45.035,-179.489,5.674,148.849
C06166=1200.126,27.400,-45.020,-179.491,5.673,148.850
C06167=1200.131,27.150,-45.005,-179.494,5.673,148.850
C06168=1200.136,26.901,-44.990,-179.497,5.672,148.851
C06169=1200.141,26.652,-44.975,-179.499,5.671,148.852
C06170=1200.146,26.402,-44.960,-179.502,5.671,148.852
C06171=1200.151,26.153,-44.945,-179.504,5.670,148.853
C06172=1200.156,25.904,-44.930,-179.507,5.670,148.854
C06173=1200.161,25.653,-44.915,-179.509,5.669,148.854
C06174=1200.166,25.404,-44.900,-179.512,5.668,148.855
C06175=1200.171,25.155,-44.885,-179.514,5.668,148.855
C06176=1200.176,24.905,-44.870,-179.517,5.667,148.856
C06177=1200.181,24.656,-44.855,-179.520,5.667,148.857
C06178=1200.186,24.407,-44.840,-179.522,5.666,148.857
C06179=1200.191,24.157,-44.825,-179.524,5.665,148.858
C06180=1200.196,23.908,-44.810,-179.527,5.665,148.859
C06181=1200.201,23.658,-44.794,-179.530,5.664,148.859
C06182=1200.206,23.408,-44.780,-179.532,5.664,148.860
C06183=1200.211,23.159,-44.765,-179.534,5.663,148.860
C06184=1200.217,22.909,-44.750,-179.537,5.662,148.861
C06185=1200.221,22.660,-44.735,-179.540,5.662,148.862
C06186=1200.227,22.410,-44.720,-179.542,5.661,148.862
C06187=1200.232,22.161,-44.705,-179.545,5.661,148.863
C06188=1200.236,21.911,-44.690,-179.547,5.660,148.864
C06189=1200.241,21.661,-44.675,-179.550,5.659,148.864
C06190=1200.246,21.412,-44.660,-179.552,5.659,148.865
C06191=1200.251,21.162,-44.646,-179.555,5.658,148.866
C06192=1200.256,20.913,-44.630,-179.558,5.658,148.866
C06193=1200.261,20.663,-44.616,-179.560,5.657,148.867
C06194=1200.266,20.414,-44.601,-179.563,5.657,148.867
C06195=1200.272,20.164,-44.586,-179.565,5.656,148.868
C06196=1200.276,19.915,-44.571,-179.568,5.656,148.869
C06197=1200.281,19.665,-44.557,-179.570,5.655,148.869
C06198=1200.286,19.416,-44.542,-179.572,5.655,148.870
C06199=1200.292,19.166,-44.527,-179.575,5.654,148.871
C06200=1200.296,18.917,-44.512,-179.577,5.654,148.871
C06201=1200.301,18.668,-44.498,-179.580,5.653,148.872
C06202=1200.307,18.418,-44.483,-179.582,5.653,148.872
C06203=1200.312,18.168,-44.468,-179.585,5.652,148.873
C06204=1200.316,17.919,-44.453,-179.588,5.652,148.874
C06205=1200.321,17.670,-44.438,-179.590,5.651,148.874
C06206=1200.327,17.420,-44.424,-179.593,5.651,148.875
C06207=1200.332,17.170,-44.409,-179.595,5.650,148.876
C06208=1200.337,16.922,-44.395,-179.598,5.649,148.876
C06209=1200.342,16.672,-44.380,-179.600,5.649,148.877
C06210=1200.347,16.423,-44.365,-179.603,5.648,148.878
C06211=1200.352,16.173,-44.351,-179.606,5.648,148.878
C06212=1200.357,15.923,-44.336,-179.608,5.647,148.879
C06213=1200.362,15.674,-44.321,-179.610,5.646,148.879
C06214=1200.367,15.424,-44.307,-179.613,5.646,148.880
C06215=1200.372,15.174,-44.293,-179.616,5.645,148.881
C06216=1200.377,14.925,-44.277,-179.618,5.645,148.882
C06217=1200.382,14.675,-44.263,-179.621,5.644,148.882
C06218=1200.387,14.426,-44.249,-179.623,5.643,148.883
C06219=1200.392,14.177,-44.234,-179.625,5.644,148.883
C06220=1200.397,13.927,-44.219,-179.628,5.643,148.884
C06221=1200.402,13.677,-44.204,-179.630,5.643,148.885
C06222=1200.407,13.427,-44.190,-179.633,5.642,148.885
C06223=1200.413,13.179,-44.176,-179.635,5.641,148.886
C06224=1200.418,12.929,-44.161,-179.638,5.641,148.887
C06225=1200.423,12.679,-44.147,-179.641,5.640,148.887
C06226=1200.428,12.430,-44.133,-179.643,5.640,148.888
C06227=1200.432,12.180,-44.118,-179.646,5.639,148.889
C06228=1200.437,11.931,-44.103,-179.648,5.638,148.889
C06229=1200.443,11.681,-44.089,-179.651,5.638,148.890
C06230=1200.448,11.431,-44.074,-179.653,5.637,148.890
C06231=1200.453,11.181,-44.060,-179.656,5.637,148.891
C06232=1200.458,10.933,-44.045,-179.659,5.636,148.892
C06233=1200.463,10.683,-44.031,-179.660,5.636,148.892
C06234=1200.468,10.434,-44.017,-179.663,5.636,148.893
C06235=1200.473,10.184,-44.003,-179.666,5.635,148.894
C06236=1200.478,9.934,-43.988,-179.668,5.635,148.894
C06237=1200.483,9.684,-43.974,-179.671,5.634,148.895
C06238=1200.487,9.435,-43.959,-179.673,5.634,148.896
C06239=1200.493,9.186,-43.945,-179.676,5.633,148.896
C06240=1200.498,8.937,-43.931,-179.678,5.632,148.897
C06241=1200.503,8.687,-43.917,-179.681,5.632,148.897
C06242=1200.509,8.437,-43.902,-179.684,5.631,148.898
C06243=1200.514,8.187,-43.887,-179.686,5.631,148.899
C06244=1200.518,7.937,-43.873,-179.688,5.630,148.899
C06245=1200.524,7.688,-43.859,-179.690,5.630,148.900
C06246=1200.529,7.439,-43.845,-179.693,5.630,148.901
C06247=1200.534,7.189,-43.831,-179.696,5.629,148.901
C06248=1200.539,6.940,-43.816,-179.698,5.629,148.902
C06249=1200.544,6.690,-43.801,-179.701,5.628,148.903
C06250=1200.549,6.441,-43.787,-179.703,5.628,148.903
C06251=1200.554,6.191,-43.773,-179.706,5.627,148.904
C06252=1200.559,5.942,-43.759,-179.709,5.627,148.905
C06253=1200.564,5.692,-43.745,-179.711,5.626,148.905
C06254=1200.569,5.442,-43.730,-179.714,5.626,148.906
C06255=1200.574,5.194,-43.717,-179.715,5.625,148.906
C06256=1200.579,4.944,-43.703,-179.718,5.625,148.907
C06257=1200.584,4.694,-43.689,-179.721,5.624,148.908
C06258=1200.589,4.445,-43.674,-179.723,5.624,148.908
C06259=1200.594,4.196,-43.660,-179.726,5.623,148.909
C06260=1200.599,3.946,-43.646,-179.729,5.623,148.910
C06261=1200.604,3.696,-43.632,-179.731,5.622,148.910
C06262=1200.609,3.446,-43.617,-179.734,5.622,148.911
C06263=1200.614,3.177,-43.602,-179.736,5.621,148.912
C06264=1200.620,2.908,-43.588,-179.739,5.621,148.912
C06265=1200.626,2.639,-43.573,-179.741,5.620,148.913
C06266=1200.631,2.370,-43.557,-179.744,5.620,148.914
C06267=1200.636,2.120,-43.543,-179.747,5.619,148.914
C06268=1200.641,1.871,-43.529,-179.749,5.619,148.915
C06269=1200.647,1.621,-43.515,-179.752,5.618,148.916
C06270=1200.652,1.371,-43.501,-179.754,5.618,148.916
C06271=1200.657,1.122,-43.487,-179.757,5.618,148.917
C06272=1200.662,0.873,-43.474,-179.759,5.617,148.918
C06273=1200.666,0.623,-43.459,-179.762,5.617,148.918
C06274=1200.671,0.373,-43.445,-179.764,5.616,148.919
C06275=1200.676,0.124,-43.431,-179.767,5.616,148.920
C06276=1200.682,-0.126,-43.418,-179.770,5.615,148.920
C06277=1200.687,-0.376,-43.403,-179.772,5.614,148.921
C06278=1200.692,-0.625,-43.389,-179.774,5.615,148.922
C06279=1200.697,-0.874,-43.376,-179.777,5.614,148.922
C06280=1200.702,-1.124,-43.361,-179.779,5.614,148.923
C06281=1200.707,-1.374,-43.348,-179.782,5.613,148.924
C06282=1200.713,-1.623,-43.334,-179.784,5.613,148.924
C06283=1200.718,-1.873,-43.320,-179.787,5.612,148.925
C06284=1200.722,-2.122,-43.306,-179.789,5.611,148.925
C06285=1200.727,-2.371,-43.292,-179.791,5.612,148.926
C06286=1200.733,-2.622,-43.278,-179.794,5.611,148.927
C06287=1200.738,-2.871,-43.264,-179.797,5.611,148.928
C06288=1200.743,-3.120,-43.250,-179.799,5.610,148.928
C06289=1200.747,-3.370,-43.237,-179.801,5.609,148.929
C06290=1200.753,-3.620,-43.223,-179.804,5.609,148.929
C06291=1200.758,-3.869,-43.209,-179.807,5.608,148.930
C06292=1200.763,-4.119,-43.195,-179.809,5.609,148.931
C06293=1200.768,-4.369,-43.182,-179.812,5.608,148.931
C06294=1200.773,-4.618,-43.168,-179.814,5.608,148.932
C06295=1200.778,-4.867,-43.154,-179.816,5.607,148.933
C06296=1200.784,-5.118,-43.140,-179.819,5.606,148.933
C06297=1200.788,-5.366,-43.127,-179.822,5.606,148.934
C06298=1200.793,-5.616,-43.113,-179.824,5.605,148.935
C06299=1200.799,-5.866,-43.099,-179.826,5.606,148.935
C06300=1200.803,-6.115,-43.086,-179.829,5.605,148.936
C06301=1200.808,-6.365,-43.071,-179.831,5.604,148.936
C06302=1200.814,-6.615,-43.058,-179.834,5.604,148.937
C06303=1200.818,-6.864,-43.045,-179.837,5.603,148.938
C06304=1200.824,-7.114,-43.031,-179.839,5.603,148.939
C06305=1200.829,-7.363,-43.017,-179.841,5.603,148.939
C06306=1200.833,-7.613,-43.003,-179.844,5.603,148.940
C06307=1200.839,-7.862,-42.990,-179.846,5.602,148.940
C06308=1200.844,-8.112,-42.976,-179.849,5.601,148.941
C06309=1200.849,-8.361,-42.963,-179.851,5.601,148.942
C06310=1200.854,-8.611,-42.949,-179.854,5.600,148.942
C06311=1200.859,-8.861,-42.935,-179.856,5.601,148.943
C06312=1200.864,-9.110,-42.922,-179.859,5.600,148.944
C06313=1200.869,-9.360,-42.908,-179.861,5.600,148.945
C06314=1200.875,-9.609,-42.895,-179.864,5.599,148.945
C06315=1200.879,-9.859,-42.881,-179.866,5.598,148.946
C06316=1200.885,-10.108,-42.868,-179.869,5.598,148.946
C06317=1200.890,-10.358,-42.854,-179.871,5.598,148.947
C06318=1200.895,-10.607,-42.841,-179.874,5.598,148.948
C06319=1200.900,-10.857,-42.827,-179.876,5.597,148.948
C06320=1200.905,-11.107,-42.814,-179.878,5.596,148.949
C06321=1200.910,-11.356,-42.800,-179.881,5.596,148.950
C06322=1200.915,-11.606,-42.787,-179.884,5.595,148.950
C06323=1200.921,-11.855,-42.773,-179.886,5.596,148.951
C06324=1200.926,-12.106,-42.759,-179.889,5.595,148.952
C06325=1200.931,-12.355,-42.747,-179.891,5.595,148.952
C06326=1200.936,-12.605,-42.732,-179.893,5.594,148.953
C06327=1200.941,-12.854,-42.720,-179.896,5.593,148.954
C06328=1200.946,-13.104,-42.706,-179.899,5.593,148.954
C06329=1200.951,-13.353,-42.693,-179.901,5.593,148.955
C06330=1200.956,-13.603,-42.679,-179.903,5.593,148.956
C06331=1200.961,-13.852,-42.666,-179.906,5.592,148.956
C06332=1200.966,-14.102,-42.653,-179.908,5.591,148.957
C06333=1200.971,-14.351,-42.639,-179.911,5.591,148.957
C06334=1200.976,-14.601,-42.626,-179.913,5.591,148.958
C06335=1200.982,-14.851,-42.612,-179.916,5.591,148.959
C06336=1200.987,-15.100,-42.599,-179.918,5.590,148.960
C06337=1200.992,-15.350,-42.586,-179.921,5.590,148.960
C06338=1200.997,-15.600,-42.573,-179.924,5.589,148.961
C06339=1201.002,-15.849,-42.559,-179.925,5.589,148.961
C06340=1201.007,-16.099,-42.546,-179.928,5.589,148.962
C06341=1201.012,-16.348,-42.533,-179.930,5.588,148.963
C06342=1201.017,-16.598,-42.519,-179.933,5.588,148.963
C06343=1201.022,-16.847,-42.506,-179.936,5.587,148.964
C06344=1201.028,-17.097,-42.493,-179.938,5.588,148.965
C06345=1201.032,-17.346,-42.479,-179.940,5.587,148.965
C06346=1201.038,-17.596,-42.466,-179.943,5.586,148.966
C06347=1201.043,-17.846,-42.453,-179.945,5.586,148.967
C06348=1201.049,-18.096,-42.440,-179.948,5.585,148.967
C06349=1201.053,-18.345,-42.426,-179.950,5.586,148.968
C06350=1201.059,-18.595,-42.413,-179.953,5.585,148.969
C06351=1201.064,-18.844,-42.401,-179.955,5.585,148.970
C06352=1201.068,-19.094,-42.388,-179.958,5.584,148.970
C06353=1201.074,-19.343,-42.374,-179.960,5.583,148.971
C06354=1201.078,-19.593,-42.361,-179.962,5.584,148.971
C06355=1201.084,-19.843,-42.347,-179.965,5.583,148.972
C06356=1201.089,-20.093,-42.335,-179.968,5.583,148.973
C06357=1201.094,-20.342,-42.322,-179.970,5.582,148.973
C06358=1201.099,-20.591,-42.308,-179.972,5.582,148.974
C06359=1201.104,-20.841,-42.295,-179.975,5.582,148.975
C06360=1201.110,-21.091,-42.282,-179.977,5.581,148.975
C06361=1201.115,-21.340,-42.269,-179.980,5.581,148.976
C06362=1201.119,-21.590,-42.256,-179.983,5.580,148.977
C06363=1201.125,-21.840,-42.243,-179.985,5.581,148.977
C06364=1201.130,-22.089,-42.229,-179.987,5.580,148.978
C06365=1201.135,-22.338,-42.217,-179.989,5.579,148.979
C06366=1201.141,-22.588,-42.204,-179.992,5.579,148.979
C06367=1201.146,-22.858,-42.190,-179.995,5.578,148.980
C06368=1201.151,-23.128,-42.176,-179.997,5.578,148.981
C06369=1201.157,-23.397,-42.162,-179.999,5.578,148.981
C06370=1201.162,-23.666,-42.147,179.998,5.578,148.982
C06371=1201.167,-23.915,-42.135,179.995,5.577,148.983
C06372=1201.173,-24.166,-42.121,179.993,5.577,148.983
C06373=1201.178,-24.415,-42.109,179.990,5.576,148.984
C06374=1201.182,-24.665,-42.096,179.988,5.577,148.985
C06375=1201.187,-24.914,-42.083,179.985,5.576,148.986
C06376=1201.193,-25.164,-42.070,179.982,5.576,148.986
C06377=1201.198,-25.414,-42.057,179.980,5.575,148.987
C06378=1201.203,-25.663,-42.044,179.978,5.575,148.987
C06379=1201.208,-25.913,-42.032,179.976,5.575,148.988
C06380=1201.213,-26.163,-42.018,179.973,5.574,148.989
C06381=1201.218,-26.412,-42.005,179.970,5.574,148.989
C06382=1201.224,-26.662,-41.993,179.968,5.573,148.990
C06383=1201.229,-26.911,-41.980,179.966,5.574,148.991
C06384=1201.234,-27.161,-41.967,179.963,5.573,148.991
C06385=1201.239,-27.411,-41.954,179.961,5.572,148.992
C06386=1201.244,-27.660,-41.942,179.958,5.572,148.993
C06387=1201.249,-27.910,-41.929,179.956,5.572,148.993
C06388=1201.255,-28.160,-41.915,179.953,5.572,148.994
C06389=1201.260,-28.409,-41.903,179.951,5.571,148.995
C06390=1201.264,-28.659,-41.890,179.948,5.571,148.995
C06391=1201.269,-28.908,-41.877,179.946,5.571,148.996
C06392=1201.274,-29.158,-41.865,179.944,5.570,148.997
C06393=1201.280,-29.407,-41.851,179.941,5.570,148.997
C06394=1201.285,-29.657,-41.838,179.938,5.569,148.998
C06395=1201.290,-29.907,-41.827,179.936,5.570,148.999
C06396=1201.295,-30.157,-41.814,179.934,5.569,148.999
C06397=1201.301,-30.406,-41.801,179.931,5.569,149.000
C06398=1201.306,-30.656,-41.788,179.929,5.568,149.001
C06399=1201.311,-30.906,-41.775,179.927,5.568,149.001
C06400=1201.316,-31.155,-41.763,179.924,5.568,149.002
C06401=1201.321,-31.404,-41.750,179.921,5.567,149.003
C06402=1201.326,-31.654,-41.737,179.919,5.567,149.003
C06403=1201.331,-31.904,-41.725,179.917,5.567,149.004
C06404=1201.336,-32.153,-41.713,179.915,5.566,149.005
C06405=1201.342,-32.403,-41.699,179.912,5.566,149.005
C06406=1201.347,-32.653,-41.686,179.909,5.566,149.006
C06407=1201.352,-32.902,-41.674,179.907,5.566,149.007
C06408=1201.357,-33.152,-41.662,179.904,5.565,149.007
C06409=1201.362,-33.402,-41.649,179.902,5.565,149.008
C06410=1201.367,-33.651,-41.637,179.900,5.565,149.009
C06411=1201.372,-33.901,-41.624,179.898,5.564,149.009
C06412=1201.377,-34.150,-41.611,179.895,5.564,149.010
C06413=1201.383,-34.400,-41.599,179.892,5.564,149.011
C06414=1201.388,-34.650,-41.587,179.890,5.564,149.011
C06415=1201.394,-34.899,-41.573,179.887,5.563,149.012
C06416=1201.398,-35.149,-41.560,179.885,5.563,149.013
C06417=1201.403,-35.399,-41.549,179.883,5.562,149.013
C06418=1201.409,-35.648,-41.536,179.881,5.562,149.014
C06419=1201.414,-35.898,-41.523,179.878,5.562,149.015
C06420=1201.419,-36.147,-41.511,179.875,5.562,149.015
C06421=1201.424,-36.398,-41.499,179.873,5.562,149.016
C06422=1201.429,-36.647,-41.486,179.870,5.561,149.017
C06423=1201.434,-36.896,-41.473,179.868,5.561,149.017
C06424=1201.439,-37.146,-41.461,179.866,5.560,149.018
C06425=1201.444,-37.396,-41.449,179.864,5.560,149.019
C06426=1201.450,-37.645,-41.436,179.861,5.560,149.019
C06427=1201.455,-37.895,-41.424,179.858,5.560,149.020
C06428=1201.460,-38.145,-41.411,179.856,5.560,149.021
C06429=1201.465,-38.394,-41.399,179.854,5.559,149.021
C06430=1201.470,-38.644,-41.387,179.851,5.559,149.022
C06431=1201.475,-38.893,-41.374,179.849,5.558,149.023
C06432=1201.481,-39.143,-41.362,179.847,5.558,149.023
C06433=1201.486,-39.393,-41.350,179.844,5.558,149.024
C06434=1201.491,-39.642,-41.337,179.841,5.558,149.025
C06435=1201.496,-39.893,-41.325,179.840,5.557,149.025
C06436=1201.501,-40.142,-41.312,179.837,5.557,149.026
C06437=1201.506,-40.392,-41.300,179.834,5.557,149.027
C06438=1201.511,-40.641,-41.288,179.832,5.556,149.027
C06439=1201.517,-40.891,-41.275,179.830,5.556,149.028
C06440=1201.522,-41.140,-41.263,179.827,5.556,149.029
C06441=1201.527,-41.390,-41.251,179.824,5.556,149.029
C06442=1201.532,-41.640,-41.239,179.823,5.555,149.030
C06443=1201.538,-41.889,-41.226,179.820,5.555,149.031
C06444=1201.542,-42.139,-41.215,179.817,5.555,149.031
C06445=1201.547,-42.389,-41.202,179.815,5.555,149.032
C06446=1201.552,-42.639,-41.190,179.813,5.554,149.033
C06447=1201.557,-42.888,-41.178,179.810,5.554,149.033
C06448=1201.563,-43.138,-41.166,179.808,5.553,149.034
C06449=1201.568,-43.387,-41.153,179.806,5.554,149.034
C06450=1201.573,-43.637,-41.141,179.803,5.553,149.035
C06451=1201.578,-43.886,-41.129,179.800,5.553,149.036
C06452=1201.584,-44.136,-41.117,179.798,5.553,149.037
C06453=1201.588,-44.385,-41.105,179.796,5.553,149.037
C06454=1201.594,-44.635,-41.093,179.793,5.552,149.038
C06455=1201.599,-44.885,-41.080,179.791,5.552,149.038
C06456=1201.604,-45.135,-41.068,179.789,5.552,149.039
C06457=1201.609,-45.384,-41.056,179.786,5.551,149.040
C06458=1201.615,-45.634,-41.044,179.783,5.551,149.041
C06459=1201.620,-45.884,-41.032,179.781,5.551,149.041
C06460=1201.625,-46.133,-41.020,179.779,5.551,149.042
C06461=1201.630,-46.383,-41.008,179.776,5.550,149.042
C06462=1201.635,-46.633,-40.995,179.774,5.550,149.043
C06463=1201.640,-46.883,-40.983,179.772,5.550,149.044
C06464=1201.645,-47.133,-40.971,179.769,5.549,149.045
C06465=1201.651,-47.382,-40.959,179.767,5.550,149.045
C06466=1201.655,-47.632,-40.947,179.764,5.549,149.046
C06467=1201.661,-47.882,-40.936,179.762,5.548,149.046
C06468=1201.666,-48.131,-40.923,179.760,5.549,149.047
C06469=1201.671,-48.381,-40.911,179.757,5.548,149.048
C06470=1201.676,-48.630,-40.898,179.755,5.548,149.049
C06471=1201.682,-48.900,-40.886,179.753,5.548,149.049
C06472=1201.688,-49.170,-40.873,179.750,5.548,149.050
C06473=1201.694,-49.440,-40.860,179.747,5.547,149.051
C06474=1201.699,-49.710,-40.847,179.745,5.547,149.051
C06475=1201.704,-49.960,-40.835,179.742,5.546,149.052
C06476=1201.709,-50.210,-40.824,179.740,5.547,149.053
C06477=1201.714,-50.459,-40.812,179.737,5.546,149.053
C06478=1201.720,-50.709,-40.800,179.734,5.546,149.054
C06479=1201.725,-50.959,-40.788,179.733,5.546,149.055
C06480=1201.729,-51.208,-40.776,179.730,5.545,149.055
C06481=1201.735,-51.458,-40.764,179.728,5.545,149.056
C06482=1201.740,-51.708,-40.752,179.725,5.545,149.057
C06483=1201.746,-51.958,-40.740,179.723,5.545,149.057
C06484=1201.750,-52.207,-40.729,179.720,5.544,149.058
C06485=1201.755,-52.457,-40.716,179.719,5.544,149.059
C06486=1201.761,-52.707,-40.704,179.716,5.544,149.059
C06487=1201.766,-52.956,-40.693,179.713,5.543,149.060
C06488=1201.771,-53.206,-40.681,179.711,5.544,149.061
C06489=1201.777,-53.455,-40.669,179.708,5.543,149.061
C06490=1201.781,-53.704,-40.658,179.706,5.543,149.062
C06491=1201.787,-53.954,-40.646,179.704,5.543,149.063
C06492=1201.792,-54.204,-40.634,179.702,5.542,149.063
C06493=1201.797,-54.454,-40.623,179.699,5.542,149.064
C06494=1201.802,-54.704,-40.611,179.697,5.542,149.065
C06495=1201.807,-54.953,-40.598,179.694,5.542,149.065
C06496=1201.812,-55.203,-40.587,179.691,5.541,149.066
C06497=1201.818,-55.453,-40.575,179.690,5.541,149.067
C06498=1201.823,-55.703,-40.563,179.687,5.541,149.067
C06499=1201.828,-55.952,-40.552,179.685,5.541,149.068
C06500=1201.833,-56.202,-40.540,179.682,5.541,149.069
C06501=1201.838,-56.451,-40.529,179.680,5.540,149.069
C06502=1201.844,-56.700,-40.516,179.678,5.541,149.070
C06503=1201.849,-56.950,-40.504,179.676,5.540,149.071
C06504=1201.854,-57.200,-40.493,179.673,5.539,149.071
C06505=1201.859,-57.450,-40.481,179.671,5.540,149.072
C06506=1201.864,-57.700,-40.470,179.668,5.539,149.073
C06507=1201.869,-57.949,-40.458,179.665,5.539,149.073
C06508=1201.874,-58.199,-40.447,179.664,5.539,149.074
C06509=1201.879,-58.449,-40.435,179.661,5.538,149.075
C06510=1201.885,-58.698,-40.423,179.659,5.538,149.075
C06511=1201.890,-58.948,-40.412,179.656,5.538,149.076
C06512=1201.896,-59.198,-40.400,179.654,5.538,149.077
C06513=1201.900,-59.447,-40.389,179.652,5.538,149.077
C06514=1201.906,-59.697,-40.377,179.650,5.537,149.078
C06515=1201.910,-59.947,-40.366,179.647,5.537,149.079
C06516=1201.916,-60.196,-40.354,179.645,5.537,149.079
C06517=1201.921,-60.446,-40.343,179.642,5.537,149.080
C06518=1201.926,-60.696,-40.331,179.639,5.536,149.081
C06519=1201.931,-60.945,-40.320,179.637,5.537,149.081
C06520=1201.937,-61.195,-40.308,179.635,5.536,149.082
C06521=1201.942,-61.445,-40.296,179.632,5.535,149.083
C06522=1201.947,-61.694,-40.285,179.630,5.536,149.083
C06523=1201.953,-61.944,-40.273,179.628,5.535,149.084
C06524=1201.957,-62.194,-40.262,179.626,5.536,149.085
C06525=1201.963,-62.444,-40.250,179.623,5.535,149.085
C06526=1201.968,-62.693,-40.239,179.621,5.534,149.086
C06527=1201.972,-62.943,-40.227,179.619,5.535,149.087
C06528=1201.978,-63.192,-40.216,179.616,5.534,149.087
C06529=1201.983,-63.442,-40.205,179.613,5.534,149.088
C06530=1201.988,-63.692,-40.193,179.611,5.534,149.089
C06531=1201.993,-63.942,-40.182,179.609,5.533,149.089
C06532=1201.999,-64.191,-40.171,179.607,5.534,149.090
C06533=1202.004,-64.441,-40.159,179.604,5.533,149.091
C06534=1202.010,-64.691,-40.147,179.602,5.533,149.091
C06535=1202.014,-64.940,-40.136,179.600,5.533,149.092
C06536=1202.020,-65.190,-40.124,179.597,5.532,149.093
C06537=1202.025,-65.439,-40.113,179.595,5.532,149.093
C06538=1202.030,-65.690,-40.103,179.593,5.532,149.094
C06539=1202.035,-65.939,-40.091,179.590,5.532,149.095
C06540=1202.040,-66.189,-40.080,179.588,5.532,149.095
C06541=1202.046,-66.438,-40.068,179.585,5.532,149.096
C06542=1202.051,-66.688,-40.057,179.583,5.531,149.097
C06543=1202.056,-66.938,-40.045,179.581,5.531,149.097
C06544=1202.061,-67.188,-40.034,179.578,5.531,149.098
C06545=1202.067,-67.437,-40.023,179.576,5.531,149.099
C06546=1202.072,-67.687,-40.012,179.574,5.531,149.099
C06547=1202.077,-67.937,-40.000,179.571,5.530,149.100
C06548=1202.081,-68.186,-39.989,179.569,5.530,149.101
C06549=1202.088,-68.436,-39.978,179.567,5.530,149.101
C06550=1202.092,-68.686,-39.967,179.564,5.530,149.102
C06551=1202.098,-68.936,-39.955,179.562,5.530,149.103
C06552=1202.103,-69.185,-39.944,179.560,5.529,149.103
C06553=1202.108,-69.435,-39.933,179.558,5.529,149.104
C06554=1202.114,-69.685,-39.922,179.555,5.529,149.105
C06555=1202.119,-69.934,-39.911,179.552,5.529,149.105
C06556=1202.124,-70.184,-39.900,179.550,5.529,149.106
C06557=1202.129,-70.434,-39.888,179.548,5.528,149.106
C06558=1202.134,-70.684,-39.877,179.546,5.529,149.107
C06559=1202.139,-70.932,-39.866,179.543,5.528,149.108
C06560=1202.145,-71.183,-39.855,179.541,5.528,149.109
C06561=1202.150,-71.433,-39.844,179.539,5.528,149.109
C06562=1202.155,-71.682,-39.833,179.536,5.528,149.110
C06563=1202.161,-71.932,-39.821,179.534,5.528,149.110
C06564=1202.165,-72.182,-39.810,179.532,5.527,149.111
C06565=1202.171,-72.431,-39.799,179.529,5.527,149.112
C06566=1202.176,-72.681,-39.789,179.527,5.527,149.113
C06567=1202.181,-72.931,-39.777,179.524,5.527,149.113
C06568=1202.186,-73.180,-39.766,179.523,5.527,149.114
C06569=1202.191,-73.430,-39.755,179.520,5.526,149.114
C06570=1202.197,-73.680,-39.743,179.517,5.526,149.115
C06571=1202.202,-73.929,-39.733,179.515,5.526,149.116
C06572=1202.207,-74.179,-39.722,179.512,5.526,149.117
C06573=1202.212,-74.428,-39.711,179.511,5.526,149.117
C06574=1202.218,-74.679,-39.700,179.508,5.525,149.118
C06575=1202.223,-74.949,-39.688,179.506,5.525,149.119
C06576=1202.229,-75.220,-39.676,179.503,5.525,149.119
C06577=1202.235,-75.491,-39.664,179.501,5.525,149.120
C06578=1202.240,-75.761,-39.652,179.498,5.524,149.121
C06579=1202.246,-76.011,-39.642,179.496,5.525,149.121
C06580=1202.251,-76.261,-39.630,179.493,5.524,149.122
C06581=1202.256,-76.511,-39.620,179.491,5.524,149.123
C06582=1202.262,-76.760,-39.608,179.489,5.524,149.123
C06583=1202.267,-77.010,-39.598,179.486,5.523,149.124
C06584=1202.272,-77.259,-39.587,179.484,5.524,149.125
C06585=1202.277,-77.509,-39.575,179.482,5.523,149.125
C06586=1202.282,-77.759,-39.565,179.480,5.524,149.126
C06587=1202.288,-78.008,-39.553,179.477,5.523,149.127
C06588=1202.293,-78.259,-39.543,179.475,5.522,149.127
C06589=1202.298,-78.508,-39.532,179.473,5.523,149.128
C06590=1202.303,-78.758,-39.521,179.470,5.522,149.129
C06591=1202.309,-79.007,-39.511,179.468,5.523,149.129
C06592=1202.313,-79.257,-39.500,179.466,5.522,149.130
C06593=1202.318,-79.507,-39.489,179.463,5.522,149.131
C06594=1202.324,-79.756,-39.478,179.461,5.522,149.131
C06595=1202.329,-80.007,-39.467,179.458,5.521,149.132
C06596=1202.335,-80.256,-39.456,179.457,5.521,149.132
C06597=1202.340,-80.506,-39.446,179.454,5.521,149.133
C06598=1202.345,-80.755,-39.435,179.452,5.521,149.134
C06599=1202.350,-81.005,-39.424,179.449,5.521,149.135
C06600=1202.355,-81.255,-39.413,179.447,5.521,149.135
C06601=1202.360,-81.504,-39.403,179.445,5.521,149.136
C06602=1202.366,-81.755,-39.391,179.442,5.520,149.137
C06603=1202.371,-82.004,-39.380,179.440,5.520,149.137
C06604=1202.376,-82.254,-39.370,179.438,5.520,149.138
C06605=1202.382,-82.503,-39.360,179.436,5.520,149.138
C06606=1202.387,-82.753,-39.348,179.433,5.520,149.139
C06607=1202.392,-83.003,-39.338,179.431,5.519,149.140
C06608=1202.397,-83.253,-39.328,179.428,5.520,149.141
C06609=1202.402,-83.502,-39.317,179.426,5.519,149.141
C06610=1202.407,-83.752,-39.306,179.424,5.519,149.142
C06611=1202.413,-84.002,-39.296,179.422,5.519,149.142
C06612=1202.418,-84.251,-39.285,179.419,5.519,149.143
C06613=1202.423,-84.501,-39.274,179.417,5.519,149.144
C06614=1202.428,-84.751,-39.264,179.415,5.519,149.144
C06615=1202.434,-85.000,-39.253,179.413,5.518,149.145
C06616=1202.439,-85.250,-39.242,179.410,5.518,149.146
C06617=1202.444,-85.500,-39.232,179.408,5.518,149.146
C06618=1202.449,-85.749,-39.221,179.405,5.518,149.147
C06619=1202.455,-85.999,-39.211,179.403,5.518,149.148
C06620=1202.460,-86.249,-39.200,179.401,5.517,149.148
C06621=1202.465,-86.499,-39.190,179.399,5.518,149.149
C06622=1202.470,-86.748,-39.179,179.396,5.517,149.150
C06623=1202.475,-86.998,-39.168,179.394,5.517,149.150
C06624=1202.480,-87.248,-39.158,179.392,5.517,149.151
C06625=1202.486,-87.498,-39.148,179.389,5.516,149.152
C06626=1202.491,-87.747,-39.136,179.387,5.517,149.152
C06627=1202.496,-87.997,-39.126,179.385,5.516,149.153
C06628=1202.501,-88.247,-39.115,179.383,5.516,149.154
C06629=1202.507,-88.497,-39.105,179.380,5.516,149.154
C06630=1202.512,-88.747,-39.095,179.378,5.516,149.155
C06631=1202.517,-88.996,-39.084,179.376,5.516,149.155
C06632=1202.523,-89.245,-39.074,179.374,5.516,149.156
C06633=1202.528,-89.496,-39.063,179.371,5.515,149.157
C06634=1202.533,-89.745,-39.053,179.368,5.515,149.158
C06635=1202.538,-89.995,-39.042,179.366,5.515,149.158
C06636=1202.544,-90.245,-39.032,179.364,5.515,149.159
C06637=1202.549,-90.495,-39.021,179.362,5.515,149.160
C06638=1202.554,-90.744,-39.010,179.359,5.515,149.160
C06639=1202.559,-90.994,-39.000,179.357,5.515,149.161
C06640=1202.565,-91.244,-38.990,179.355,5.514,149.161
C06641=1202.570,-91.493,-38.979,179.353,5.515,149.162
C06642=1202.575,-91.743,-38.970,179.350,5.514,149.163
C06643=1202.580,-91.993,-38.959,179.348,5.515,149.164
C06644=1202.585,-92.243,-38.949,179.346,5.514,149.164
C06645=1202.591,-92.492,-38.938,179.344,5.514,149.165
C06646=1202.596,-92.742,-38.928,179.341,5.514,149.165
C06647=1202.601,-92.992,-38.917,179.339,5.513,149.166
C06648=1202.607,-93.241,-38.907,179.337,5.513,149.167
C06649=1202.612,-93.492,-38.896,179.334,5.513,149.167
C06650=1202.617,-93.741,-38.887,179.332,5.513,149.168
C06651=1202.622,-93.990,-38.876,179.330,5.513,149.169
C06652=1202.627,-94.241,-38.866,179.328,5.513,149.169
C06653=1202.633,-94.490,-38.856,179.325,5.512,149.170
C06654=1202.638,-94.740,-38.845,179.323,5.513,149.171
C06655=1202.643,-94.990,-38.835,179.321,5.512,149.171
C06656=1202.649,-95.240,-38.825,179.319,5.512,149.172
C06657=1202.654,-95.489,-38.815,179.316,5.512,149.173
C06658=1202.659,-95.739,-38.804,179.314,5.512,149.173
C06659=1202.665,-95.989,-38.794,179.312,5.511,149.174
C06660=1202.670,-96.239,-38.784,179.309,5.511,149.175
C06661=1202.675,-96.488,-38.773,179.307,5.511,149.175
C06662=1202.681,-96.738,-38.763,179.305,5.511,149.176
C06663=1202.685,-96.988,-38.753,179.303,5.511,149.176
C06664=1202.691,-97.237,-38.743,179.300,5.511,149.177
C06665=1202.696,-97.487,-38.733,179.298,5.511,149.178
C06666=1202.701,-97.737,-38.722,179.295,5.511,149.179
C06667=1202.707,-97.987,-38.712,179.294,5.511,149.179
C06668=1202.712,-98.236,-38.702,179.291,5.510,149.180
C06669=1202.717,-98.486,-38.692,179.289,5.511,149.180
C06670=1202.722,-98.736,-38.682,179.286,5.510,149.181
C06671=1202.728,-98.985,-38.671,179.285,5.510,149.182
C06672=1202.733,-99.234,-38.662,179.282,5.510,149.182
C06673=1202.738,-99.485,-38.652,179.280,5.510,149.183
C06674=1202.744,-99.735,-38.642,179.278,5.509,149.184
C06675=1202.749,-99.984,-38.632,179.276,5.510,149.184
C06676=1202.753,-100.234,-38.622,179.273,5.509,149.185
C06677=1202.759,-100.484,-38.611,179.271,5.510,149.186
C06678=1202.765,-100.733,-38.601,179.269,5.509,149.186
C06679=1202.770,-101.005,-38.590,179.266,5.508,149.187
C06680=1202.776,-101.277,-38.579,179.264,5.509,149.188
C06681=1202.782,-101.548,-38.569,179.261,5.508,149.188
C06682=1202.787,-101.819,-38.558,179.259,5.508,149.189
C06683=1202.793,-102.068,-38.548,179.257,5.508,149.190
C06684=1202.798,-102.319,-38.537,179.254,5.508,149.190
C06685=1202.803,-102.569,-38.528,179.252,5.508,149.191
C06686=1202.808,-102.818,-38.518,179.250,5.508,149.192
C06687=1202.813,-103.068,-38.507,179.248,5.508,149.192
C06688=1202.818,-103.318,-38.498,179.245,5.508,149.193
C06689=1202.824,-103.567,-38.488,179.243,5.508,149.194
C06690=1202.829,-103.817,-38.477,179.241,5.507,149.194
C06691=1202.834,-104.067,-38.468,179.239,5.508,149.195
C06692=1202.840,-104.317,-38.458,179.236,5.507,149.196
C06693=1202.845,-104.566,-38.448,179.234,5.507,149.196
C06694=1202.850,-104.815,-38.438,179.232,5.507,149.197
C06695=1202.855,-105.066,-38.428,179.230,5.507,149.197
C06696=1202.861,-105.316,-38.418,179.227,5.506,149.198
C06697=1202.866,-105.565,-38.408,179.225,5.507,149.199
C06698=1202.871,-105.815,-38.398,179.223,5.506,149.200
C06699=1202.877,-106.065,-38.389,179.221,5.506,149.200
C06700=1202.882,-106.315,-38.379,179.218,5.506,149.201
C06701=1202.887,-106.564,-38.369,179.216,5.506,149.201
C06702=1202.892,-106.814,-38.359,179.214,5.505,149.202
C06703=1202.898,-107.064,-38.349,179.212,5.506,149.203
C06704=1202.903,-107.314,-38.339,179.209,5.505,149.203
C06705=1202.908,-107.563,-38.329,179.207,5.506,149.204
C06706=1202.914,-107.813,-38.320,179.205,5.505,149.205
C06707=1202.919,-108.063,-38.310,179.203,5.505,149.205
C06708=1202.924,-108.312,-38.300,179.200,5.505,149.206
C06709=1202.929,-108.563,-38.291,179.199,5.505,149.206
C06710=1202.934,-108.812,-38.280,179.196,5.505,149.207
C06711=1202.940,-109.062,-38.270,179.194,5.505,149.208
C06712=1202.945,-109.312,-38.261,179.192,5.504,149.208
C06713=1202.951,-109.561,-38.251,179.190,5.505,149.209
C06714=1202.956,-109.810,-38.242,179.187,5.504,149.210
C06715=1202.961,-110.061,-38.232,179.185,5.504,149.210
C06716=1202.966,-110.310,-38.222,179.183,5.504,149.211
C06717=1202.972,-110.561,-38.213,179.181,5.504,149.212
C06718=1202.976,-110.810,-38.203,179.178,5.504,149.212
C06719=1202.982,-111.059,-38.193,179.176,5.504,149.213
C06720=1202.988,-111.310,-38.183,179.174,5.503,149.214
C06721=1202.992,-111.560,-38.173,179.172,5.504,149.214
C06722=1202.998,-111.810,-38.164,179.169,5.503,149.215
C06723=1203.003,-112.059,-38.154,179.167,5.503,149.216
C06724=1203.009,-112.309,-38.145,179.165,5.503,149.216
C06725=1203.014,-112.558,-38.135,179.163,5.503,149.217
C06726=1203.019,-112.808,-38.125,179.160,5.503,149.218
C06727=1203.025,-113.058,-38.116,179.158,5.503,149.218
C06728=1203.030,-113.307,-38.106,179.156,5.502,149.219
C06729=1203.035,-113.558,-38.096,179.154,5.503,149.219
C06730=1203.040,-113.807,-38.086,179.151,5.502,149.220
C06731=1203.045,-114.057,-38.077,179.150,5.502,149.221
C06732=1203.050,-114.306,-38.068,179.147,5.502,149.221
C06733=1203.056,-114.557,-38.058,179.145,5.502,149.222
C06734=1203.061,-114.806,-38.049,179.143,5.502,149.223
C06735=1203.067,-115.056,-38.039,179.141,5.502,149.223
C06736=1203.072,-115.305,-38.030,179.139,5.502,149.224
C06737=1203.078,-115.555,-38.020,179.136,5.501,149.224
C06738=1203.082,-115.805,-38.010,179.134,5.502,149.225
C06739=1203.088,-116.055,-38.001,179.132,5.501,149.226
C06740=1203.093,-116.305,-37.991,179.130,5.501,149.226
C06741=1203.099,-116.555,-37.981,179.127,5.501,149.227
C06742=1203.104,-116.805,-37.973,179.125,5.501,149.228
C06743=1203.109,-117.054,-37.963,179.123,5.501,149.228
C06744=1203.115,-117.304,-37.953,179.121,5.501,149.229
C06745=1203.119,-117.553,-37.944,179.118,5.501,149.230
C06746=1203.125,-117.803,-37.934,179.117,5.501,149.230
C06747=1203.130,-118.053,-37.925,179.114,5.500,149.231
C06748=1203.135,-118.303,-37.916,179.112,5.501,149.232
C06749=1203.141,-118.553,-37.906,179.110,5.500,149.232
C06750=1203.146,-118.802,-37.897,179.108,5.500,149.233
C06751=1203.151,-119.053,-37.887,179.105,5.500,149.234
C06752=1203.156,-119.302,-37.877,179.103,5.500,149.234
C06753=1203.162,-119.552,-37.868,179.101,5.499,149.235
C06754=1203.167,-119.802,-37.859,179.099,5.500,149.235
C06755=1203.172,-120.051,-37.849,179.096,5.499,149.236
C06756=1203.177,-120.301,-37.840,179.094,5.499,149.237
C06757=1203.183,-120.551,-37.831,179.092,5.500,149.237
C06758=1203.188,-120.801,-37.821,179.090,5.499,149.238
C06759=1203.193,-121.050,-37.812,179.088,5.499,149.239
C06760=1203.199,-121.301,-37.803,179.086,5.499,149.239
C06761=1203.204,-121.550,-37.793,179.084,5.499,149.240
C06762=1203.209,-121.800,-37.784,179.081,5.499,149.241
C06763=1203.215,-122.050,-37.775,179.079,5.499,149.241
C06764=1203.220,-122.299,-37.765,179.077,5.498,149.242
C06765=1203.225,-122.549,-37.756,179.075,5.499,149.242
C06766=1203.231,-122.799,-37.747,179.072,5.498,149.243
C06767=1203.236,-123.048,-37.737,179.070,5.498,149.244
C06768=1203.241,-123.298,-37.728,179.068,5.498,149.244
C06769=1203.246,-123.548,-37.719,179.066,5.498,149.245
C06770=1203.252,-123.798,-37.710,179.063,5.497,149.246
C06771=1203.257,-124.047,-37.700,179.062,5.497,149.246
C06772=1203.262,-124.297,-37.691,179.059,5.497,149.247
C06773=1203.268,-124.547,-37.682,179.057,5.497,149.247
C06774=1203.273,-124.797,-37.673,179.055,5.497,149.248
C06775=1203.278,-125.046,-37.663,179.053,5.497,149.249
C06776=1203.283,-125.296,-37.655,179.051,5.497,149.249
C06777=1203.289,-125.547,-37.645,179.048,5.497,149.250
C06778=1203.294,-125.796,-37.636,179.046,5.497,149.251
C06779=1203.300,-126.046,-37.627,179.044,5.496,149.251
C06780=1203.304,-126.295,-37.618,179.042,5.497,149.252
C06781=1203.310,-126.546,-37.608,179.039,5.496,149.253
C06782=1203.316,-126.795,-37.599,179.038,5.496,149.253
C06783=1202.894,-126.806,-37.637,179.033,5.500,149.255
C06784=1202.889,-126.557,-37.647,179.035,5.500,149.254
C06785=1202.884,-126.307,-37.656,179.038,5.500,149.254
C06786=1202.878,-126.057,-37.665,179.040,5.500,149.253
C06787=1202.873,-125.807,-37.674,179.042,5.500,149.252
C06788=1202.868,-125.557,-37.683,179.044,5.500,149.252
C06789=1202.863,-125.308,-37.693,179.047,5.501,149.251
C06790=1202.857,-125.057,-37.702,179.049,5.500,149.251
C06791=1202.852,-124.808,-37.711,179.051,5.501,149.250
C06792=1202.847,-124.558,-37.720,179.053,5.501,149.249
C06793=1202.841,-124.308,-37.729,179.056,5.501,149.249
C06794=1202.836,-124.058,-37.739,179.057,5.501,149.248
C06795=1202.831,-123.809,-37.748,179.059,5.501,149.247
C06796=1202.825,-123.559,-37.757,179.062,5.501,149.247
C06797=1202.820,-123.309,-37.767,179.064,5.501,149.246
C06798=1202.815,-123.059,-37.776,179.066,5.501,149.245
C06799=1202.810,-122.809,-37.785,179.068,5.501,149.245
C06800=1202.804,-122.559,-37.794,179.071,5.502,149.244
C06801=1202.799,-122.310,-37.804,179.073,5.501,149.244
C06802=1202.794,-122.060,-37.813,179.075,5.502,149.243
C06803=1202.788,-121.810,-37.822,179.077,5.502,149.242
C06804=1202.783,-121.561,-37.832,179.080,5.502,149.242
C06805=1202.778,-121.311,-37.841,179.081,5.502,149.241
C06806=1202.773,-121.061,-37.850,179.084,5.503,149.240
C06807=1202.767,-120.812,-37.860,179.086,5.503,149.240
C06808=1202.762,-120.562,-37.869,179.088,5.503,149.239
C06809=1202.757,-120.312,-37.878,179.090,5.503,149.239
C06810=1202.751,-120.062,-37.888,179.093,5.503,149.238
C06811=1202.746,-119.812,-37.897,179.095,5.503,149.237
C06812=1202.741,-119.563,-37.906,179.097,5.503,149.237
C06813=1202.735,-119.313,-37.916,179.099,5.503,149.236
C06814=1202.730,-119.063,-37.925,179.101,5.503,149.235
C06815=1202.724,-118.813,-37.934,179.104,5.503,149.235
C06816=1202.719,-118.564,-37.944,179.105,5.503,149.234
C06817=1202.714,-118.314,-37.953,179.108,5.504,149.233
C06818=1202.708,-118.064,-37.963,179.110,5.503,149.233
C06819=1202.703,-117.815,-37.972,179.112,5.504,149.232
C06820=1202.699,-117.564,-37.981,179.114,5.504,149.232
C06821=1202.693,-117.314,-37.992,179.117,5.504,149.231
C06822=1202.688,-117.065,-38.000,179.119,5.504,149.230
C06823=1202.682,-116.815,-38.011,179.121,5.505,149.230
C06824=1202.677,-116.565,-38.020,179.123,5.505,149.229
C06825=1202.672,-116.316,-38.030,179.126,5.505,149.228
C06826=1202.666,-116.066,-38.039,179.128,5.505,149.228
C06827=1202.661,-115.817,-38.048,179.130,5.505,149.227
C06828=1202.656,-115.566,-38.058,179.132,5.505,149.227
C06829=1202.650,-115.317,-38.067,179.135,5.505,149.226
C06830=1202.645,-115.067,-38.077,179.136,5.505,149.225
C06831=1202.640,-114.817,-38.086,179.139,5.506,149.225
C06832=1202.635,-114.567,-38.096,179.141,5.505,149.224
C06833=1202.629,-114.317,-38.105,179.143,5.506,149.223
C06834=1202.624,-114.068,-38.115,179.145,5.506,149.223
C06835=1202.619,-113.818,-38.124,179.148,5.506,149.222
C06836=1202.613,-113.568,-38.135,179.149,5.506,149.222
C06837=1202.608,-113.318,-38.143,179.152,5.507,149.221
C06838=1202.603,-113.069,-38.153,179.154,5.506,149.220
C06839=1202.598,-112.820,-38.163,179.156,5.506,149.219
C06840=1202.592,-112.570,-38.172,179.159,5.507,149.219
C06841=1202.587,-112.319,-38.183,179.161,5.506,149.218
C06842=1202.582,-112.070,-38.192,179.163,5.507,149.217
C06843=1202.577,-111.820,-38.202,179.165,5.507,149.217
C06844=1202.571,-111.570,-38.211,179.168,5.507,149.216
C06845=1202.566,-111.321,-38.221,179.170,5.507,149.216
C06846=1202.560,-111.070,-38.230,179.172,5.507,149.215
C06847=1202.555,-110.821,-38.240,179.174,5.507,149.214
C06848=1202.550,-110.571,-38.251,179.177,5.507,149.214
C06849=1202.545,-110.321,-38.260,179.178,5.507,149.213
C06850=1202.539,-110.072,-38.270,179.181,5.508,149.212
C06851=1202.534,-109.822,-38.279,179.183,5.507,149.212
C06852=1202.529,-109.572,-38.289,179.185,5.508,149.211
C06853=1202.524,-109.323,-38.298,179.187,5.508,149.211
C06854=1202.518,-109.072,-38.308,179.190,5.508,149.210
C06855=1202.513,-108.823,-38.318,179.192,5.508,149.209
C06856=1202.508,-108.573,-38.328,179.194,5.509,149.209
C06857=1202.502,-108.323,-38.338,179.196,5.508,149.208
C06858=1202.497,-108.074,-38.347,179.199,5.509,149.207
C06859=1202.492,-107.824,-38.358,179.201,5.509,149.207
C06860=1202.487,-107.574,-38.367,179.203,5.509,149.206
C06861=1202.481,-107.324,-38.377,179.205,5.509,149.205
C06862=1202.476,-107.075,-38.387,179.208,5.509,149.205
C06863=1202.471,-106.825,-38.396,179.210,5.509,149.204
C06864=1202.466,-106.575,-38.407,179.212,5.509,149.203
C06865=1202.461,-106.325,-38.416,179.214,5.509,149.203
C06866=1202.455,-106.076,-38.426,179.217,5.510,149.202
C06867=1202.449,-105.826,-38.436,179.219,5.509,149.201
C06868=1202.444,-105.576,-38.446,179.221,5.510,149.201
C06869=1202.439,-105.326,-38.456,179.223,5.510,149.200
C06870=1202.435,-105.077,-38.466,179.226,5.510,149.200
C06871=1202.429,-104.827,-38.475,179.228,5.510,149.199
C06872=1202.423,-104.577,-38.485,179.230,5.511,149.198
C06873=1202.419,-104.327,-38.495,179.232,5.510,149.198
C06874=1202.413,-104.078,-38.506,179.235,5.511,149.197
C06875=1202.407,-103.828,-38.515,179.236,5.511,149.196
C06876=1202.402,-103.578,-38.525,179.239,5.511,149.196
C06877=1202.397,-103.328,-38.535,179.242,5.512,149.195
C06878=1202.392,-103.079,-38.545,179.244,5.511,149.194
C06879=1202.387,-102.829,-38.555,179.246,5.512,149.194
C06880=1202.381,-102.579,-38.565,179.248,5.512,149.193
C06881=1202.376,-102.329,-38.575,179.251,5.512,149.192
C06882=1202.371,-102.080,-38.585,179.252,5.512,149.192
C06883=1202.366,-101.830,-38.595,179.255,5.512,149.191
C06884=1202.360,-101.559,-38.606,179.257,5.512,149.190
C06885=1202.354,-101.287,-38.617,179.260,5.512,149.190
C06886=1202.348,-101.016,-38.627,179.262,5.513,149.189
C06887=1202.342,-100.745,-38.639,179.264,5.512,149.188
C06888=1202.338,-100.495,-38.648,179.267,5.513,149.188
C06889=1202.333,-100.245,-38.659,179.269,5.513,149.187
C06890=1202.327,-99.995,-38.669,179.271,5.513,149.186
C06891=1202.322,-99.746,-38.678,179.273,5.513,149.186
C06892=1202.317,-99.495,-38.689,179.276,5.513,149.185
C06893=1202.311,-99.246,-38.699,179.278,5.513,149.184
C06894=1202.306,-98.996,-38.709,179.280,5.514,149.184
C06895=1202.301,-98.746,-38.719,179.283,5.513,149.183
C06896=1202.296,-98.497,-38.729,179.285,5.514,149.183
C06897=1202.290,-98.247,-38.740,179.287,5.514,149.182
C06898=1202.285,-97.997,-38.750,179.289,5.514,149.181
C06899=1202.280,-97.747,-38.760,179.292,5.514,149.180
C06900=1202.275,-97.498,-38.770,179.294,5.515,149.180
C06901=1202.270,-97.248,-38.781,179.296,5.514,149.179
C06902=1202.264,-96.998,-38.791,179.299,5.515,149.179
C06903=1202.259,-96.749,-38.801,179.301,5.515,149.178
C06904=1202.254,-96.499,-38.811,179.303,5.515,149.177
C06905=1202.248,-96.249,-38.820,179.305,5.515,149.177
C06906=1202.243,-95.999,-38.831,179.308,5.515,149.176
C06907=1202.238,-95.749,-38.841,179.310,5.515,149.175
C06908=1202.232,-95.499,-38.851,179.312,5.515,149.175
C06909=1202.227,-95.250,-38.862,179.315,5.516,149.174
C06910=1202.222,-95.000,-38.873,179.317,5.515,149.173
C06911=1202.217,-94.751,-38.882,179.319,5.516,149.173
C06912=1202.211,-94.502,-38.893,179.321,5.516,149.172
C06913=1202.206,-94.251,-38.903,179.324,5.516,149.171
C06914=1202.201,-94.002,-38.913,179.326,5.516,149.171
C06915=1202.195,-93.752,-38.924,179.328,5.517,149.170
C06916=1202.190,-93.502,-38.934,179.330,5.516,149.169
C06917=1202.185,-93.253,-38.944,179.333,5.517,149.169
C06918=1202.180,-93.002,-38.954,179.335,5.517,149.168
C06919=1202.175,-92.753,-38.965,179.337,5.517,149.168
C06920=1202.169,-92.503,-38.975,179.340,5.518,149.167
C06921=1202.164,-92.253,-38.985,179.342,5.517,149.166
C06922=1202.159,-92.004,-38.996,179.344,5.518,149.165
C06923=1202.154,-91.753,-39.006,179.346,5.518,149.165
C06924=1202.148,-91.504,-39.016,179.349,5.518,149.164
C06925=1202.143,-91.255,-39.027,179.351,5.518,149.164
C06926=1202.138,-91.005,-39.038,179.353,5.518,149.163
C06927=1202.133,-90.755,-39.048,179.355,5.518,149.162
C06928=1202.128,-90.505,-39.058,179.358,5.519,149.162
C06929=1202.122,-90.256,-39.068,179.360,5.519,149.161
C06930=1202.117,-90.005,-39.079,179.362,5.519,149.160
C06931=1202.112,-89.756,-39.089,179.365,5.519,149.160
C06932=1202.106,-89.507,-39.100,179.367,5.519,149.159
C06933=1202.101,-89.257,-39.111,179.369,5.519,149.158
C06934=1202.096,-89.007,-39.121,179.371,5.519,149.158
C06935=1202.091,-88.757,-39.131,179.374,5.520,149.157
C06936=1202.085,-88.507,-39.142,179.376,5.519,149.156
C06937=1202.080,-88.258,-39.153,179.378,5.520,149.156
C06938=1202.075,-88.008,-39.163,179.380,5.520,149.155
C06939=1202.070,-87.758,-39.174,179.383,5.520,149.154
C06940=1202.064,-87.508,-39.184,179.385,5.521,149.154
C06941=1202.059,-87.259,-39.194,179.387,5.520,149.153
C06942=1202.054,-87.009,-39.205,179.390,5.521,149.152
C06943=1202.048,-86.760,-39.216,179.392,5.520,149.152
C06944=1202.043,-86.509,-39.226,179.394,5.521,149.151
C06945=1202.038,-86.260,-39.236,179.396,5.521,149.150
C06946=1202.033,-86.010,-39.248,179.399,5.521,149.150
C06947=1202.027,-85.761,-39.258,179.401,5.521,149.149
C06948=1202.022,-85.510,-39.268,179.403,5.522,149.149
C06949=1202.017,-85.261,-39.279,179.406,5.522,149.148
C06950=1202.012,-85.011,-39.290,179.408,5.522,149.147
C06951=1202.007,-84.762,-39.300,179.411,5.522,149.146
C06952=1202.002,-84.512,-39.311,179.412,5.522,149.146
C06953=1201.996,-84.263,-39.322,179.415,5.523,149.145
C06954=1201.991,-84.012,-39.332,179.417,5.522,149.145
C06955=1201.986,-83.763,-39.342,179.420,5.523,149.144
C06956=1201.981,-83.513,-39.354,179.422,5.523,149.143
C06957=1201.975,-83.264,-39.364,179.424,5.523,149.143
C06958=1201.970,-83.013,-39.375,179.427,5.524,149.142
C06959=1201.965,-82.764,-39.385,179.429,5.523,149.141
C06960=1201.960,-82.514,-39.396,179.431,5.524,149.140
C06961=1201.955,-82.264,-39.407,179.433,5.524,149.140
C06962=1201.950,-82.015,-39.418,179.436,5.524,149.139
C06963=1201.945,-81.765,-39.428,179.438,5.524,149.139
C06964=1201.939,-81.516,-39.440,179.441,5.524,149.138
C06965=1201.934,-81.265,-39.450,179.443,5.525,149.137
C06966=1201.928,-81.016,-39.460,179.445,5.524,149.137
C06967=1201.924,-80.766,-39.472,179.447,5.525,149.136
C06968=1201.918,-80.517,-39.482,179.450,5.525,149.135
C06969=1201.913,-80.267,-39.493,179.452,5.525,149.135
C06970=1201.908,-80.017,-39.503,179.454,5.525,149.134
C06971=1201.903,-79.767,-39.514,179.456,5.525,149.133
C06972=1201.897,-79.517,-39.526,179.459,5.526,149.133
C06973=1201.892,-79.268,-39.536,179.461,5.525,149.132
C06974=1201.887,-79.018,-39.547,179.464,5.526,149.131
C06975=1201.881,-78.769,-39.558,179.465,5.526,149.131
C06976=1201.877,-78.519,-39.569,179.468,5.526,149.130
C06977=1201.871,-78.269,-39.579,179.471,5.527,149.129
C06978=1201.866,-78.020,-39.590,179.473,5.526,149.129
C06979=1201.861,-77.769,-39.602,179.475,5.527,149.128
C06980=1201.855,-77.520,-39.612,179.477,5.527,149.127
C06981=1201.850,-77.270,-39.623,179.480,5.527,149.127
C06982=1201.845,-77.021,-39.634,179.482,5.527,149.126
C06983=1201.840,-76.771,-39.645,179.485,5.527,149.125
C06984=1201.835,-76.521,-39.656,179.487,5.528,149.125
C06985=1201.829,-76.271,-39.667,179.489,5.528,149.124
C06986=1201.824,-76.022,-39.678,179.492,5.528,149.123
C06987=1201.819,-75.772,-39.688,179.494,5.528,149.123
C06988=1201.813,-75.501,-39.700,179.496,5.528,149.122
C06989=1201.807,-75.230,-39.713,179.499,5.529,149.121
C06990=1201.801,-74.960,-39.724,179.502,5.529,149.121
C06991=1201.796,-74.689,-39.736,179.504,5.529,149.120
C06992=1201.791,-74.439,-39.748,179.506,5.529,149.119
C06993=1201.785,-74.190,-39.758,179.508,5.529,149.119
C06994=1201.781,-73.940,-39.770,179.511,5.530,149.118
C06995=1201.776,-73.690,-39.780,179.513,5.530,149.117
C06996=1201.770,-73.441,-39.792,179.515,5.530,149.117
C06997=1201.765,-73.191,-39.803,179.518,5.530,149.116
C06998=1201.759,-72.942,-39.813,179.520,5.530,149.115
C06999=1201.755,-72.692,-39.824,179.522,5.531,149.115
C07000=1201.749,-72.441,-39.836,179.525,5.531,149.114
C07001=1201.744,-72.192,-39.847,179.527,5.531,149.113
C07002=1201.739,-71.943,-39.858,179.530,5.531,149.113
C07003=1201.733,-71.692,-39.869,179.531,5.531,149.112
C07004=1201.728,-71.443,-39.880,179.534,5.532,149.111
C07005=1201.723,-71.194,-39.891,179.537,5.532,149.111
C07006=1201.717,-70.943,-39.902,179.539,5.532,149.110
C07007=1201.712,-70.694,-39.913,179.542,5.532,149.109
C07008=1201.708,-70.445,-39.925,179.543,5.532,149.109
C07009=1201.702,-70.195,-39.936,179.546,5.532,149.108
C07010=1201.697,-69.944,-39.947,179.548,5.533,149.107
C07011=1201.692,-69.696,-39.958,179.551,5.533,149.107
C07012=1201.686,-69.446,-39.970,179.553,5.533,149.106
C07013=1201.681,-69.195,-39.980,179.555,5.533,149.105
C07014=1201.676,-68.946,-39.991,179.557,5.533,149.105
C07015=1201.671,-68.696,-40.003,179.560,5.534,149.104
C07016=1201.666,-68.447,-40.015,179.562,5.534,149.103
C07017=1201.661,-68.197,-40.025,179.565,5.534,149.103
C07018=1201.655,-67.947,-40.037,179.567,5.535,149.102
C07019=1201.650,-67.698,-40.048,179.569,5.534,149.101
C07020=1201.646,-67.448,-40.059,179.572,5.535,149.101
C07021=1201.639,-67.198,-40.070,179.574,5.534,149.100
C07022=1201.635,-66.949,-40.081,179.577,5.535,149.099
C07023=1201.629,-66.699,-40.093,179.579,5.536,149.099
C07024=1201.624,-66.449,-40.104,179.581,5.535,149.098
C07025=1201.619,-66.200,-40.115,179.584,5.536,149.097
C07026=1201.614,-65.950,-40.127,179.586,5.535,149.097
C07027=1201.609,-65.700,-40.138,179.588,5.536,149.096
C07028=1201.603,-65.450,-40.150,179.591,5.536,149.095
C07029=1201.598,-65.201,-40.161,179.593,5.536,149.095
C07030=1201.593,-64.951,-40.173,179.595,5.537,149.094
C07031=1201.588,-64.702,-40.184,179.598,5.537,149.093
C07032=1201.583,-64.452,-40.195,179.600,5.537,149.093
C07033=1201.578,-64.202,-40.207,179.603,5.537,149.092
C07034=1201.572,-63.952,-40.217,179.604,5.537,149.092
C07035=1201.567,-63.703,-40.229,179.607,5.538,149.091
C07036=1201.562,-63.453,-40.240,179.610,5.538,149.090
C07037=1201.557,-63.203,-40.252,179.612,5.538,149.089
C07038=1201.551,-62.954,-40.263,179.614,5.538,149.089
C07039=1201.546,-62.704,-40.275,179.617,5.539,149.088
C07040=1201.541,-62.454,-40.286,179.619,5.539,149.088
C07041=1201.536,-62.205,-40.298,179.621,5.539,149.087
C07042=1201.531,-61.955,-40.310,179.623,5.539,149.086
C07043=1201.525,-61.706,-40.321,179.626,5.539,149.085
C07044=1201.520,-61.456,-40.332,179.629,5.540,149.085
C07045=1201.515,-61.206,-40.344,179.630,5.540,149.084
C07046=1201.510,-60.956,-40.356,179.633,5.540,149.084
C07047=1201.505,-60.707,-40.367,179.636,5.541,149.083
C07048=1201.500,-60.457,-40.379,179.638,5.540,149.082
C07049=1201.494,-60.207,-40.390,179.640,5.541,149.081
C07050=1201.489,-59.957,-40.401,179.643,5.541,149.081
C07051=1201.484,-59.708,-40.413,179.645,5.541,149.080
C07052=1201.479,-59.458,-40.425,179.647,5.542,149.080
C07053=1201.474,-59.209,-40.437,179.649,5.541,149.079
C07054=1201.469,-58.959,-40.448,179.652,5.542,149.078
C07055=1201.464,-58.709,-40.460,179.655,5.542,149.077
C07056=1201.458,-58.460,-40.471,179.656,5.542,149.077
C07057=1201.453,-58.210,-40.483,179.659,5.543,149.076
C07058=1201.448,-57.960,-40.494,179.662,5.543,149.076
C07059=1201.443,-57.711,-40.506,179.664,5.543,149.075
C07060=1201.437,-57.461,-40.518,179.666,5.543,149.074
C07061=1201.433,-57.211,-40.529,179.669,5.544,149.073
C07062=1201.427,-56.961,-40.541,179.671,5.544,149.073
C07063=1201.422,-56.711,-40.553,179.673,5.544,149.072
C07064=1201.417,-56.462,-40.564,179.676,5.545,149.072
C07065=1201.411,-56.212,-40.575,179.678,5.544,149.071
C07066=1201.406,-55.963,-40.587,179.681,5.545,149.070
C07067=1201.401,-55.713,-40.599,179.683,5.544,149.069
C07068=1201.396,-55.463,-40.611,179.685,5.545,149.069
C07069=1201.391,-55.214,-40.623,179.688,5.546,149.068
C07070=1201.386,-54.964,-40.634,179.690,5.545,149.068
C07071=1201.380,-54.714,-40.646,179.692,5.546,149.067
C07072=1201.376,-54.464,-40.658,179.695,5.546,149.066
C07073=1201.370,-54.214,-40.670,179.697,5.546,149.066
C07074=1201.365,-53.965,-40.682,179.699,5.547,149.065
C07075=1201.360,-53.716,-40.693,179.702,5.547,149.064
C07076=1201.354,-53.466,-40.705,179.704,5.547,149.064
C07077=1201.349,-53.216,-40.717,179.707,5.547,149.063
C07078=1201.344,-52.967,-40.728,179.709,5.548,149.062
C07079=1201.339,-52.717,-40.741,179.711,5.548,149.062
C07080=1201.334,-52.467,-40.753,179.714,5.548,149.061
C07081=1201.329,-52.218,-40.764,179.716,5.548,149.060
C07082=1201.324,-51.968,-40.776,179.718,5.548,149.060
C07083=1201.318,-51.718,-40.788,179.721,5.549,149.059
C07084=1201.314,-51.469,-40.800,179.724,5.549,149.058
C07085=1201.308,-51.219,-40.812,179.725,5.549,149.058
C07086=1201.303,-50.969,-40.823,179.728,5.549,149.057
C07087=1201.298,-50.720,-40.836,179.731,5.550,149.056
C07088=1201.293,-50.470,-40.847,179.733,5.550,149.056
C07089=1201.288,-50.220,-40.859,179.735,5.550,149.055
C07090=1201.282,-49.970,-40.871,179.738,5.550,149.054
C07091=1201.277,-49.721,-40.884,179.740,5.550,149.054
C07092=1201.271,-49.451,-40.896,179.742,5.551,149.053
C07093=1201.266,-49.181,-40.909,179.745,5.551,149.052
C07094=1201.261,-48.910,-40.922,179.748,5.551,149.051
C07095=1201.255,-48.641,-40.935,179.751,5.552,149.051
C07096=1201.249,-48.391,-40.947,179.753,5.552,149.050
C07097=1201.244,-48.142,-40.959,179.755,5.552,149.049
C07098=1201.239,-47.892,-40.971,179.758,5.553,149.049
C07099=1201.234,-47.642,-40.982,179.760,5.553,149.048
C07100=1201.229,-47.393,-40.995,179.762,5.553,149.047
C07101=1201.223,-47.143,-41.007,179.765,5.553,149.047
C07102=1201.218,-46.893,-41.019,179.767,5.553,149.046
C07103=1201.214,-46.644,-41.031,179.769,5.554,149.045
C07104=1201.208,-46.394,-41.043,179.772,5.554,149.045
C07105=1201.203,-46.145,-41.055,179.774,5.554,149.044
C07106=1201.198,-45.895,-41.067,179.777,5.554,149.043
C07107=1201.192,-45.645,-41.079,179.779,5.555,149.043
C07108=1201.187,-45.395,-41.092,179.782,5.555,149.042
C07109=1201.182,-45.146,-41.103,179.784,5.555,149.041
C07110=1201.178,-44.896,-41.116,179.786,5.556,149.041
C07111=1201.172,-44.646,-41.128,179.789,5.556,149.040
C07112=1201.167,-44.396,-41.140,179.791,5.556,149.039
C07113=1201.162,-44.147,-41.152,179.794,5.556,149.039
C07114=1201.157,-43.897,-41.165,179.796,5.557,149.038
C07115=1201.151,-43.647,-41.177,179.798,5.557,149.038
C07116=1201.147,-43.398,-41.188,179.801,5.557,149.037
C07117=1201.141,-43.148,-41.201,179.803,5.558,149.036
C07118=1201.136,-42.898,-41.213,179.805,5.557,149.035
C07119=1201.131,-42.649,-41.225,179.808,5.558,149.035
C07120=1201.126,-42.399,-41.237,179.811,5.558,149.034
C07121=1201.120,-42.150,-41.250,179.813,5.559,149.034
C07122=1201.115,-41.900,-41.262,179.815,5.559,149.033
C07123=1201.110,-41.651,-41.274,179.818,5.559,149.032
C07124=1201.105,-41.401,-41.287,179.820,5.560,149.031
C07125=1201.100,-41.151,-41.299,179.822,5.559,149.031
C07126=1201.095,-40.901,-41.312,179.825,5.560,149.030
C07127=1201.090,-40.652,-41.323,179.827,5.561,149.030
C07128=1201.085,-40.402,-41.336,179.830,5.561,149.029
C07129=1201.080,-40.152,-41.347,179.832,5.561,149.028
C07130=1201.074,-39.903,-41.360,179.835,5.561,149.027
C07131=1201.069,-39.654,-41.373,179.837,5.562,149.027
C07132=1201.064,-39.404,-41.384,179.839,5.561,149.026
C07133=1201.059,-39.154,-41.397,179.842,5.562,149.025
C07134=1201.054,-38.904,-41.409,179.844,5.563,149.025
C07135=1201.049,-38.655,-41.422,179.846,5.562,149.024
C07136=1201.044,-38.405,-41.435,179.849,5.563,149.023
C07137=1201.038,-38.155,-41.446,179.852,5.563,149.023
C07138=1201.033,-37.906,-41.459,179.854,5.564,149.022
C07139=1201.028,-37.657,-41.472,179.856,5.563,149.021
C07140=1201.023,-37.406,-41.484,179.859,5.564,149.021
C07141=1201.018,-37.157,-41.496,179.861,5.565,149.020
C07142=1201.013,-36.907,-41.509,179.864,5.565,149.020
C07143=1201.007,-36.657,-41.521,179.866,5.565,149.019
C07144=1201.002,-36.408,-41.534,179.869,5.565,149.018
C07145=1200.997,-36.159,-41.546,179.871,5.566,149.017
C07146=1200.992,-35.909,-41.558,179.873,5.566,149.017
C07147=1200.987,-35.659,-41.572,179.876,5.566,149.016
C07148=1200.981,-35.409,-41.584,179.878,5.567,149.016
C07149=1200.976,-35.159,-41.596,179.881,5.567,149.015
C07150=1200.971,-34.910,-41.609,179.883,5.567,149.014
C07151=1200.966,-34.661,-41.621,179.886,5.567,149.013
C07152=1200.961,-34.411,-41.634,179.888,5.568,149.013
C07153=1200.956,-34.161,-41.646,179.890,5.568,149.012
C07154=1200.951,-33.911,-41.659,179.893,5.568,149.012
C07155=1200.946,-33.662,-41.671,179.895,5.569,149.011
C07156=1200.940,-33.413,-41.684,179.898,5.569,149.010
C07157=1200.936,-33.163,-41.697,179.900,5.569,149.009
C07158=1200.930,-32.913,-41.709,179.903,5.569,149.009
C07159=1200.925,-32.663,-41.722,179.905,5.570,149.008
C07160=1200.919,-32.414,-41.735,179.908,5.571,149.008
C07161=1200.914,-32.165,-41.747,179.910,5.570,149.007
C07162=1200.910,-31.915,-41.760,179.912,5.571,149.006
C07163=1200.904,-31.665,-41.772,179.915,5.571,149.006
C07164=1200.899,-31.415,-41.785,179.918,5.572,149.005
C07165=1200.894,-31.166,-41.797,179.920,5.571,149.004
C07166=1200.889,-30.916,-41.811,179.922,5.572,149.004
C07167=1200.884,-30.666,-41.823,179.924,5.573,149.003
C07168=1200.879,-30.417,-41.836,179.927,5.573,149.002
C07169=1200.873,-30.168,-41.849,179.929,5.573,149.002
C07170=1200.869,-29.917,-41.861,179.932,5.573,149.001
C07171=1200.864,-29.668,-41.873,179.935,5.574,149.000
C07172=1200.858,-29.418,-41.887,179.937,5.575,149.000
C07173=1200.853,-29.169,-41.899,179.939,5.574,148.999
C07174=1200.848,-28.919,-41.912,179.941,5.575,148.998
C07175=1200.843,-28.669,-41.925,179.944,5.575,148.998
C07176=1200.838,-28.420,-41.937,179.947,5.576,148.997
C07177=1200.833,-28.170,-41.951,179.949,5.575,148.996
C07178=1200.827,-27.920,-41.964,179.951,5.576,148.996
C07179=1200.822,-27.671,-41.976,179.954,5.577,148.995
C07180=1200.817,-27.422,-41.989,179.956,5.577,148.994
C07181=1200.813,-27.172,-42.002,179.958,5.577,148.994
C07182=1200.807,-26.922,-42.015,179.961,5.577,148.993
C07183=1200.802,-26.673,-42.028,179.964,5.578,148.992
C07184=1200.797,-26.423,-42.041,179.966,5.578,148.992
C07185=1200.792,-26.174,-42.053,179.968,5.578,148.991
C07186=1200.786,-25.924,-42.066,179.971,5.579,148.990
C07187=1200.782,-25.674,-42.079,179.973,5.579,148.990
C07188=1200.776,-25.425,-42.092,179.976,5.580,148.989
C07189=1200.771,-25.175,-42.104,179.978,5.579,148.988
C07190=1200.766,-24.925,-42.118,179.981,5.580,148.988
C07191=1200.761,-24.676,-42.131,179.983,5.581,148.987
C07192=1200.756,-24.426,-42.143,179.986,5.581,148.986
C07193=1200.751,-24.176,-42.157,179.988,5.582,148.986
C07194=1200.745,-23.927,-42.169,179.990,5.581,148.985
C07195=1200.740,-23.677,-42.182,179.993,5.582,148.984
C07196=1200.735,-23.407,-42.196,179.996,5.582,148.984
C07197=1200.730,-23.138,-42.211,179.998,5.583,148.983
C07198=1200.724,-22.869,-42.225,-179.999,5.583,148.982
C07199=1200.719,-22.599,-42.238,-179.996,5.584,148.982
C07200=1200.713,-22.349,-42.252,-179.994,5.584,148.981
C07201=1200.708,-22.099,-42.264,-179.992,5.584,148.980
C07202=1200.703,-21.850,-42.277,-179.989,5.584,148.979
C07203=1200.698,-21.600,-42.291,-179.987,5.585,148.979
C07204=1200.693,-21.351,-42.304,-179.984,5.586,148.978
C07205=1200.688,-21.102,-42.317,-179.982,5.585,148.978
C07206=1200.683,-20.851,-42.330,-179.979,5.586,148.977
C07207=1200.677,-20.602,-42.343,-179.977,5.586,148.976
C07208=1200.672,-20.352,-42.356,-179.974,5.587,148.976
C07209=1200.667,-20.103,-42.369,-179.971,5.587,148.975
C07210=1200.662,-19.854,-42.382,-179.970,5.587,148.974
C07211=1200.657,-19.603,-42.396,-179.967,5.588,148.974
C07212=1200.652,-19.354,-42.408,-179.965,5.588,148.973
C07213=1200.647,-19.104,-42.422,-179.962,5.589,148.972
C07214=1200.642,-18.855,-42.435,-179.959,5.589,148.972
C07215=1200.637,-18.606,-42.448,-179.957,5.589,148.971
C07216=1200.631,-18.355,-42.461,-179.955,5.590,148.970
C07217=1200.626,-18.106,-42.474,-179.952,5.590,148.970
C07218=1200.621,-17.856,-42.488,-179.950,5.591,148.969
C07219=1200.616,-17.607,-42.501,-179.947,5.591,148.968
C07220=1200.611,-17.357,-42.514,-179.945,5.591,148.968
C07221=1200.606,-17.107,-42.527,-179.942,5.591,148.967
C07222=1200.600,-16.858,-42.541,-179.940,5.592,148.967
C07223=1200.596,-16.608,-42.554,-179.937,5.592,148.966
C07224=1200.590,-16.359,-42.567,-179.935,5.593,148.965
C07225=1200.586,-16.109,-42.581,-179.933,5.593,148.964
C07226=1200.581,-15.860,-42.593,-179.930,5.593,148.964
C07227=1200.575,-15.610,-42.607,-179.927,5.594,148.963
C07228=1200.570,-15.360,-42.620,-179.925,5.594,148.962
C07229=1200.565,-15.111,-42.634,-179.923,5.595,148.962
C07230=1200.560,-14.861,-42.646,-179.921,5.595,148.961
C07231=1200.555,-14.612,-42.661,-179.918,5.595,148.960
C07232=1200.550,-14.362,-42.673,-179.915,5.596,148.960
C07233=1200.545,-14.112,-42.687,-179.913,5.596,148.959
C07234=1200.539,-13.863,-42.701,-179.910,5.596,148.958
C07235=1200.535,-13.613,-42.714,-179.908,5.597,148.958
C07236=1200.529,-13.363,-42.727,-179.906,5.597,148.957
C07237=1200.525,-13.114,-42.741,-179.903,5.598,148.957
C07238=1200.519,-12.864,-42.754,-179.900,5.598,148.956
C07239=1200.515,-12.615,-42.767,-179.898,5.598,148.955
C07240=1200.509,-12.365,-42.781,-179.895,5.599,148.954
C07241=1200.504,-12.116,-42.794,-179.893,5.599,148.954
C07242=1200.499,-11.866,-42.808,-179.891,5.599,148.953
C07243=1200.494,-11.616,-42.821,-179.888,5.600,148.953
C07244=1200.489,-11.367,-42.834,-179.885,5.600,148.952
C07245=1200.483,-11.117,-42.848,-179.883,5.601,148.951
C07246=1200.478,-10.868,-42.861,-179.881,5.601,148.951
C07247=1200.473,-10.618,-42.875,-179.879,5.601,148.950
C07248=1200.468,-10.369,-42.888,-179.876,5.602,148.949
C07249=1200.463,-10.119,-42.902,-179.873,5.602,148.949
C07250=1200.458,-9.869,-42.916,-179.871,5.603,148.948
C07251=1200.453,-9.620,-42.929,-179.868,5.603,148.947
C07252=1200.448,-9.370,-42.943,-179.866,5.603,148.947
C07253=1200.443,-9.121,-42.955,-179.864,5.604,148.946
C07254=1200.438,-8.871,-42.970,-179.861,5.604,148.945
C07255=1200.432,-8.622,-42.984,-179.858,5.605,148.945
C07256=1200.428,-8.372,-42.997,-179.856,5.605,148.944
C07257=1200.423,-8.122,-43.011,-179.853,5.606,148.943
C07258=1200.417,-7.873,-43.024,-179.851,5.606,148.943
C07259=1200.413,-7.623,-43.038,-179.849,5.606,148.942
C07260=1200.407,-7.374,-43.051,-179.846,5.607,148.942
C07261=1200.402,-7.124,-43.065,-179.844,5.607,148.941
C07262=1200.398,-6.875,-43.079,-179.841,5.608,148.940
C07263=1200.392,-6.625,-43.092,-179.838,5.608,148.939
C07264=1200.387,-6.375,-43.106,-179.836,5.609,148.939
C07265=1200.382,-6.126,-43.119,-179.834,5.609,148.938
C07266=1200.377,-5.876,-43.133,-179.831,5.609,148.938
C07267=1200.372,-5.627,-43.148,-179.829,5.610,148.937
C07268=1200.366,-5.377,-43.161,-179.826,5.610,148.936
C07269=1200.362,-5.128,-43.174,-179.823,5.611,148.936
C07270=1200.356,-4.879,-43.188,-179.821,5.611,148.935
C07271=1200.351,-4.628,-43.202,-179.819,5.611,148.934
C07272=1200.347,-4.379,-43.216,-179.816,5.612,148.934
C07273=1200.341,-4.130,-43.230,-179.814,5.612,148.933
C07274=1200.336,-3.879,-43.243,-179.811,5.613,148.932
C07275=1200.331,-3.630,-43.257,-179.808,5.613,148.932
C07276=1200.326,-3.381,-43.271,-179.806,5.614,148.931
C07277=1200.321,-3.131,-43.285,-179.804,5.615,148.931
C07278=1200.316,-2.881,-43.299,-179.802,5.614,148.930
C07279=1200.311,-2.632,-43.312,-179.799,5.615,148.929
C07280=1200.306,-2.382,-43.327,-179.796,5.615,148.928
C07281=1200.301,-2.132,-43.340,-179.794,5.616,148.928
C07282=1200.295,-1.883,-43.354,-179.791,5.616,148.927
C07283=1200.291,-1.634,-43.368,-179.789,5.617,148.927
C07284=1200.286,-1.384,-43.382,-179.786,5.618,148.926
C07285=1200.280,-1.135,-43.396,-179.783,5.618,148.925
C07286=1200.275,-0.885,-43.409,-179.781,5.618,148.925
C07287=1200.271,-0.635,-43.423,-179.779,5.618,148.924
C07288=1200.265,-0.386,-43.437,-179.776,5.619,148.923
C07289=1200.260,-0.136,-43.451,-179.774,5.620,148.923
C07290=1200.255,0.113,-43.466,-179.771,5.620,148.922
C07291=1200.249,0.363,-43.479,-179.769,5.621,148.921
C07292=1200.245,0.612,-43.493,-179.766,5.621,148.921
C07293=1200.240,0.862,-43.507,-179.763,5.622,148.920
C07294=1200.235,1.112,-43.521,-179.761,5.621,148.919
C07295=1200.230,1.361,-43.535,-179.759,5.622,148.919
C07296=1200.225,1.610,-43.549,-179.756,5.623,148.918
C07297=1200.220,1.860,-43.564,-179.754,5.623,148.917
C07298=1200.214,2.109,-43.578,-179.751,5.624,148.917
C07299=1200.209,2.360,-43.591,-179.748,5.624,148.916
C07300=1200.204,2.628,-43.607,-179.746,5.625,148.915
C07301=1200.198,2.898,-43.622,-179.743,5.625,148.915
C07302=1200.193,3.167,-43.637,-179.741,5.626,148.914
C07303=1200.187,3.435,-43.652,-179.738,5.626,148.913
C07304=1200.182,3.685,-43.666,-179.735,5.627,148.913
C07305=1200.178,3.934,-43.680,-179.733,5.628,148.912
C07306=1200.173,4.184,-43.694,-179.730,5.628,148.911
C07307=1200.167,4.434,-43.708,-179.728,5.629,148.911
C07308=1200.162,4.683,-43.722,-179.726,5.628,148.910
C07309=1200.157,4.933,-43.736,-179.723,5.629,148.909
C07310=1200.152,5.183,-43.750,-179.720,5.629,148.909
C07311=1200.147,5.433,-43.765,-179.718,5.630,148.908
C07312=1200.142,5.682,-43.779,-179.716,5.631,148.908
